LIN {X 75.422,Y -35.957,Z -72.523,A -90.000,B 90.000,C 0.000} C_DIS
LIN {X 75.798,Y -35.942,Z -72.914,A -90.000,B 90.000,C 0.000} C_DIS
LIN {X 76.219,Y -35.930,Z -73.360,A -90.000,B 90.000,C 0.000} C_DIS
LIN {X 76.678,Y -35.924,Z -73.869,A -90.000,B 90.000,C 0.000} C_DIS
LIN {X 76.731,Y -35.865,Z -73.840,A -90.000,B 90.000,C 0.000} C_DIS
LIN {X 76.810,Y -35.794,Z -73.827,A -90.000,B 90.000,C 0.000} C_DIS
LIN {X 76.846,Y -35.765,Z -73.824,A -90.000,B 90.000,C 0.000} C_DIS
LIN {X 77.170,Y -35.545,Z -73.872,A -90.000,B 90.000,C 0.000} C_DIS
LIN {X 77.258,Y -35.499,Z -73.909,A -90.000,B 90.000,C 0.000} C_DIS
LIN {X 77.415,Y -35.431,Z -73.994,A -90.000,B 90.000,C 0.000} C_DIS
LIN {X 77.609,Y -35.368,Z -74.129,A -90.000,B 90.000,C 0.000} C_DIS
LIN {X 77.655,Y -35.356,Z -74.166,A -90.000,B 90.000,C 0.000} C_DIS
LIN {X 77.754,Y -35.347,Z -73.596,A -90.000,B 90.000,C 0.000} C_DIS
LIN {X 77.829,Y -35.339,Z -73.246,A -90.000,B 90.000,C 0.000} C_DIS
LIN {X 78.002,Y -35.325,Z -72.470,A -90.000,B 90.000,C 0.000} C_DIS
LIN {X 78.095,Y -35.319,Z -72.097,A -90.000,B 90.000,C 0.000} C_DIS
LIN {X 78.171,Y -35.317,Z -71.800,A -90.000,B 90.000,C 0.000} C_DIS
LIN {X 78.247,Y -35.314,Z -71.562,A -90.000,B 90.000,C 0.000} C_DIS
LIN {X 78.534,Y -35.309,Z -70.687,A -90.000,B 90.000,C 0.000} C_DIS
LIN {X 78.778,Y -35.308,Z -69.955,A -90.000,B 90.000,C 0.000} C_DIS
LIN {X 78.789,Y -36.719,Z -69.922,A -90.000,B 90.000,C 0.000} C_DIS
LIN {X 78.791,Y -36.729,Z -69.917,A -90.000,B 90.000,C 0.000} C_DIS
LIN {X 78.792,Y -36.756,Z -69.913,A -90.000,B 90.000,C 0.000} C_DIS
LIN {X 78.804,Y -35.308,Z -69.881,A -90.000,B 90.000,C 0.000} C_DIS
LIN {X 79.057,Y -35.310,Z -69.150,A -90.000,B 90.000,C 0.000} C_DIS
LIN {X 79.142,Y -35.308,Z -68.907,A -90.000,B 90.000,C 0.000} C_DIS
LIN {X 79.365,Y -35.304,Z -68.248,A -90.000,B 90.000,C 0.000} C_DIS
LIN {X 79.416,Y -35.303,Z -68.080,A -90.000,B 90.000,C 0.000} C_DIS
LIN {X 79.428,Y -35.303,Z -68.032,A -90.000,B 90.000,C 0.000} C_DIS
LIN {X 79.454,Y -35.306,Z -67.989,A -90.000,B 90.000,C 0.000} C_DIS
LIN {X 79.532,Y -35.307,Z -67.831,A -90.000,B 90.000,C 0.000} C_DIS
LIN {X 79.818,Y -35.308,Z -67.197,A -90.000,B 90.000,C 0.000} C_DIS
LIN {X 79.922,Y -35.308,Z -66.959,A -90.000,B 90.000,C 0.000} C_DIS
LIN {X 79.922,Y -60.000,Z -66.959,A -90.000,B 90.000,C 0.000} C_DIS
LIN {X 89.581,Y -60.000,Z -54.050,A -90.000,B 90.000,C 0.000} C_DIS
LIN {X 89.581,Y -35.308,Z -54.050,A -90.000,B 90.000,C 0.000} C_DIS
LIN {X 89.698,Y -35.308,Z -53.943,A -90.000,B 90.000,C 0.000} C_DIS
LIN {X 89.987,Y -35.308,Z -53.665,A -90.000,B 90.000,C 0.000} C_DIS
LIN {X 90.272,Y -35.308,Z -53.420,A -90.000,B 90.000,C 0.000} C_DIS
LIN {X 91.215,Y -35.306,Z -52.572,A -90.000,B 90.000,C 0.000} C_DIS
LIN {X 91.916,Y -35.303,Z -51.957,A -90.000,B 90.000,C 0.000} C_DIS
LIN {X 92.305,Y -35.300,Z -51.627,A -90.000,B 90.000,C 0.000} C_DIS
LIN {X 92.595,Y -35.296,Z -51.392,A -90.000,B 90.000,C 0.000} C_DIS
LIN {X 92.801,Y -35.293,Z -51.238,A -90.000,B 90.000,C 0.000} C_DIS
LIN {X 92.938,Y -35.289,Z -51.149,A -90.000,B 90.000,C 0.000} C_DIS
LIN {X 92.966,Y -35.286,Z -51.121,A -90.000,B 90.000,C 0.000} C_DIS
LIN {X 92.990,Y -35.285,Z -51.107,A -90.000,B 90.000,C 0.000} C_DIS
LIN {X 92.992,Y -46.259,Z -51.106,A -90.000,B 90.000,C 0.000} C_DIS
LIN {X 92.993,Y -46.306,Z -51.106,A -90.000,B 90.000,C 0.000} C_DIS
LIN {X 93.018,Y -46.533,Z -51.097,A -90.000,B 90.000,C 0.000} C_DIS
LIN {X 93.039,Y -46.657,Z -51.092,A -90.000,B 90.000,C 0.000} C_DIS
LIN {X 93.071,Y -46.842,Z -51.092,A -90.000,B 90.000,C 0.000} C_DIS
LIN {X 93.093,Y -46.989,Z -51.102,A -90.000,B 90.000,C 0.000} C_DIS
LIN {X 93.119,Y -47.185,Z -51.127,A -90.000,B 90.000,C 0.000} C_DIS
LIN {X 93.133,Y -47.246,Z -51.132,A -90.000,B 90.000,C 0.000} C_DIS
LIN {X 93.143,Y -47.273,Z -51.131,A -90.000,B 90.000,C 0.000} C_DIS
LIN {X 93.155,Y -47.296,Z -51.128,A -90.000,B 90.000,C 0.000} C_DIS
LIN {X 93.171,Y -47.316,Z -51.121,A -90.000,B 90.000,C 0.000} C_DIS
LIN {X 93.191,Y -47.332,Z -51.111,A -90.000,B 90.000,C 0.000} C_DIS
LIN {X 93.215,Y -47.345,Z -51.095,A -90.000,B 90.000,C 0.000} C_DIS
LIN {X 93.244,Y -47.355,Z -51.075,A -90.000,B 90.000,C 0.000} C_DIS
LIN {X 93.279,Y -47.360,Z -51.049,A -90.000,B 90.000,C 0.000} C_DIS
LIN {X 93.321,Y -47.361,Z -51.017,A -90.000,B 90.000,C 0.000} C_DIS
LIN {X 93.424,Y -47.351,Z -50.931,A -90.000,B 90.000,C 0.000} C_DIS
LIN {X 93.559,Y -47.320,Z -50.814,A -90.000,B 90.000,C 0.000} C_DIS
LIN {X 93.733,Y -47.264,Z -50.658,A -90.000,B 90.000,C 0.000} C_DIS
LIN {X 93.948,Y -47.178,Z -50.461,A -90.000,B 90.000,C 0.000} C_DIS
LIN {X 94.208,Y -47.057,Z -50.218,A -90.000,B 90.000,C 0.000} C_DIS
LIN {X 94.519,Y -46.887,Z -49.925,A -90.000,B 90.000,C 0.000} C_DIS
LIN {X 94.884,Y -46.660,Z -49.576,A -90.000,B 90.000,C 0.000} C_DIS
LIN {X 95.309,Y -46.351,Z -49.169,A -90.000,B 90.000,C 0.000} C_DIS
LIN {X 95.545,Y -46.143,Z -48.941,A -90.000,B 90.000,C 0.000} C_DIS
LIN {X 95.670,Y -46.013,Z -48.821,A -90.000,B 90.000,C 0.000} C_DIS
LIN {X 95.798,Y -45.845,Z -48.697,A -90.000,B 90.000,C 0.000} C_DIS
LIN {X 95.864,Y -45.722,Z -48.633,A -90.000,B 90.000,C 0.000} C_DIS
LIN {X 95.897,Y -45.614,Z -48.601,A -90.000,B 90.000,C 0.000} C_DIS
LIN {X 95.904,Y -45.562,Z -48.595,A -90.000,B 90.000,C 0.000} C_DIS
LIN {X 95.906,Y -35.302,Z -48.593,A -90.000,B 90.000,C 0.000} C_DIS
LIN {X 96.069,Y -35.303,Z -48.437,A -90.000,B 90.000,C 0.000} C_DIS
LIN {X 96.365,Y -35.308,Z -48.166,A -90.000,B 90.000,C 0.000} C_DIS
LIN {X 96.504,Y -35.310,Z -48.031,A -90.000,B 90.000,C 0.000} C_DIS
LIN {X 96.976,Y -35.308,Z -47.573,A -90.000,B 90.000,C 0.000} C_DIS
LIN {X 96.976,Y -60.000,Z -47.573,A -90.000,B 90.000,C 0.000} C_DIS
LIN {X -13.596,Y -60.000,Z -67.623,A -90.000,B 90.000,C 0.000} C_DIS
LIN {X -13.596,Y -35.308,Z -67.623,A -90.000,B 90.000,C 0.000} C_DIS
LIN {X -12.574,Y -35.360,Z -67.585,A -90.000,B 90.000,C 0.000} C_DIS
LIN {X -12.388,Y -35.371,Z -67.585,A -90.000,B 90.000,C 0.000} C_DIS
LIN {X -11.858,Y -35.405,Z -67.599,A -90.000,B 90.000,C 0.000} C_DIS
LIN {X -11.441,Y -35.437,Z -67.609,A -90.000,B 90.000,C 0.000} C_DIS
LIN {X -10.549,Y -35.505,Z -67.647,A -90.000,B 90.000,C 0.000} C_DIS
LIN {X -8.614,Y -35.635,Z -67.743,A -90.000,B 90.000,C 0.000} C_DIS
LIN {X -8.402,Y -35.650,Z -67.760,A -90.000,B 90.000,C 0.000} C_DIS
LIN {X -7.555,Y -35.711,Z -67.851,A -90.000,B 90.000,C 0.000} C_DIS
LIN {X -6.626,Y -35.780,Z -67.956,A -90.000,B 90.000,C 0.000} C_DIS
LIN {X -5.314,Y -35.895,Z -68.093,A -90.000,B 90.000,C 0.000} C_DIS
LIN {X -4.465,Y -35.968,Z -68.175,A -90.000,B 90.000,C 0.000} C_DIS
LIN {X -4.298,Y -35.983,Z -68.196,A -90.000,B 90.000,C 0.000} C_DIS
LIN {X -3.714,Y -36.037,Z -68.287,A -90.000,B 90.000,C 0.000} C_DIS
LIN {X -2.584,Y -36.140,Z -68.444,A -90.000,B 90.000,C 0.000} C_DIS
LIN {X -2.065,Y -36.205,Z -68.510,A -90.000,B 90.000,C 0.000} C_DIS
LIN {X -1.663,Y -36.251,Z -68.557,A -90.000,B 90.000,C 0.000} C_DIS
LIN {X -0.777,Y -36.350,Z -68.643,A -90.000,B 90.000,C 0.000} C_DIS
LIN {X 0.304,Y -36.461,Z -68.748,A -90.000,B 90.000,C 0.000} C_DIS
LIN {X 0.445,Y -36.476,Z -68.766,A -90.000,B 90.000,C 0.000} C_DIS
LIN {X 1.033,Y -36.542,Z -68.853,A -90.000,B 90.000,C 0.000} C_DIS
LIN {X 1.072,Y -36.545,Z -68.853,A -90.000,B 90.000,C 0.000} C_DIS
LIN {X 1.180,Y -36.530,Z -68.728,A -90.000,B 90.000,C 0.000} C_DIS
LIN {X 1.354,Y -36.514,Z -68.541,A -90.000,B 90.000,C 0.000} C_DIS
LIN {X 1.487,Y -36.499,Z -68.410,A -90.000,B 90.000,C 0.000} C_DIS
LIN {X 1.693,Y -36.460,Z -68.221,A -90.000,B 90.000,C 0.000} C_DIS
LIN {X 1.761,Y -36.448,Z -68.160,A -90.000,B 90.000,C 0.000} C_DIS
LIN {X 1.873,Y -36.431,Z -68.070,A -90.000,B 90.000,C 0.000} C_DIS
LIN {X 2.044,Y -36.406,Z -67.940,A -90.000,B 90.000,C 0.000} C_DIS
LIN {X 2.234,Y -36.380,Z -67.806,A -90.000,B 90.000,C 0.000} C_DIS
LIN {X 2.406,Y -36.357,Z -67.692,A -90.000,B 90.000,C 0.000} C_DIS
LIN {X 2.639,Y -36.329,Z -67.546,A -90.000,B 90.000,C 0.000} C_DIS
LIN {X 2.812,Y -36.305,Z -67.428,A -90.000,B 90.000,C 0.000} C_DIS
LIN {X 3.276,Y -36.201,Z -67.126,A -90.000,B 90.000,C 0.000} C_DIS
LIN {X 3.444,Y -36.166,Z -67.024,A -90.000,B 90.000,C 0.000} C_DIS
LIN {X 3.614,Y -36.134,Z -66.931,A -90.000,B 90.000,C 0.000} C_DIS
LIN {X 3.853,Y -36.097,Z -66.819,A -90.000,B 90.000,C 0.000} C_DIS
LIN {X 3.948,Y -36.084,Z -66.778,A -90.000,B 90.000,C 0.000} C_DIS
LIN {X 4.233,Y -36.047,Z -66.662,A -90.000,B 90.000,C 0.000} C_DIS
LIN {X 4.353,Y -36.033,Z -66.617,A -90.000,B 90.000,C 0.000} C_DIS
LIN {X 4.683,Y -36.009,Z -66.505,A -90.000,B 90.000,C 0.000} C_DIS
LIN {X 4.875,Y -35.985,Z -66.444,A -90.000,B 90.000,C 0.000} C_DIS
LIN {X 5.852,Y -35.847,Z -66.145,A -90.000,B 90.000,C 0.000} C_DIS
LIN {X 6.202,Y -35.800,Z -66.046,A -90.000,B 90.000,C 0.000} C_DIS
LIN {X 6.435,Y -35.772,Z -65.986,A -90.000,B 90.000,C 0.000} C_DIS
LIN {X 6.689,Y -35.747,Z -65.930,A -90.000,B 90.000,C 0.000} C_DIS
LIN {X 6.738,Y -35.742,Z -65.921,A -90.000,B 90.000,C 0.000} C_DIS
LIN {X 7.225,Y -35.706,Z -65.832,A -90.000,B 90.000,C 0.000} C_DIS
LIN {X 7.523,Y -35.685,Z -65.777,A -90.000,B 90.000,C 0.000} C_DIS
LIN {X 7.613,Y -35.680,Z -65.763,A -90.000,B 90.000,C 0.000} C_DIS
LIN {X 7.872,Y -35.669,Z -65.728,A -90.000,B 90.000,C 0.000} C_DIS
LIN {X 8.114,Y -35.663,Z -65.702,A -90.000,B 90.000,C 0.000} C_DIS
LIN {X 8.854,Y -35.619,Z -65.637,A -90.000,B 90.000,C 0.000} C_DIS
LIN {X 9.243,Y -35.584,Z -65.608,A -90.000,B 90.000,C 0.000} C_DIS
LIN {X 9.497,Y -35.559,Z -65.590,A -90.000,B 90.000,C 0.000} C_DIS
LIN {X 9.712,Y -35.542,Z -65.579,A -90.000,B 90.000,C 0.000} C_DIS
LIN {X 9.853,Y -35.535,Z -65.579,A -90.000,B 90.000,C 0.000} C_DIS
LIN {X 10.047,Y -35.527,Z -65.583,A -90.000,B 90.000,C 0.000} C_DIS
LIN {X 10.154,Y -35.524,Z -65.588,A -90.000,B 90.000,C 0.000} C_DIS
LIN {X 10.498,Y -35.522,Z -65.612,A -90.000,B 90.000,C 0.000} C_DIS
LIN {X 10.799,Y -35.527,Z -65.640,A -90.000,B 90.000,C 0.000} C_DIS
LIN {X 10.993,Y -35.530,Z -65.659,A -90.000,B 90.000,C 0.000} C_DIS
LIN {X 11.036,Y -35.530,Z -65.664,A -90.000,B 90.000,C 0.000} C_DIS
LIN {X 11.092,Y -35.487,Z -65.606,A -90.000,B 90.000,C 0.000} C_DIS
LIN {X 11.178,Y -35.423,Z -65.522,A -90.000,B 90.000,C 0.000} C_DIS
LIN {X 11.344,Y -35.308,Z -65.374,A -90.000,B 90.000,C 0.000} C_DIS
LIN {X 11.344,Y -60.000,Z -65.374,A -90.000,B 90.000,C 0.000} C_DIS
LIN {X -10.557,Y -60.000,Z -65.654,A -90.000,B 90.000,C 0.000} C_DIS
LIN {X -10.557,Y -35.308,Z -65.654,A -90.000,B 90.000,C 0.000} C_DIS
LIN {X -10.015,Y -35.339,Z -65.681,A -90.000,B 90.000,C 0.000} C_DIS
LIN {X -8.500,Y -35.403,Z -65.760,A -90.000,B 90.000,C 0.000} C_DIS
LIN {X -8.411,Y -35.409,Z -65.774,A -90.000,B 90.000,C 0.000} C_DIS
LIN {X -8.173,Y -35.418,Z -65.786,A -90.000,B 90.000,C 0.000} C_DIS
LIN {X -7.110,Y -35.475,Z -65.905,A -90.000,B 90.000,C 0.000} C_DIS
LIN {X -6.382,Y -35.515,Z -65.989,A -90.000,B 90.000,C 0.000} C_DIS
LIN {X -6.093,Y -35.531,Z -66.021,A -90.000,B 90.000,C 0.000} C_DIS
LIN {X -5.091,Y -35.594,Z -66.128,A -90.000,B 90.000,C 0.000} C_DIS
LIN {X -4.180,Y -35.637,Z -66.223,A -90.000,B 90.000,C 0.000} C_DIS
LIN {X -3.966,Y -35.649,Z -66.253,A -90.000,B 90.000,C 0.000} C_DIS
LIN {X -3.387,Y -35.686,Z -66.345,A -90.000,B 90.000,C 0.000} C_DIS
LIN {X -2.118,Y -35.760,Z -66.529,A -90.000,B 90.000,C 0.000} C_DIS
LIN {X -1.766,Y -35.791,Z -66.576,A -90.000,B 90.000,C 0.000} C_DIS
LIN {X -1.433,Y -35.819,Z -66.618,A -90.000,B 90.000,C 0.000} C_DIS
LIN {X 0.371,Y -35.957,Z -66.806,A -90.000,B 90.000,C 0.000} C_DIS
LIN {X 0.430,Y -35.942,Z -66.757,A -90.000,B 90.000,C 0.000} C_DIS
LIN {X 0.581,Y -35.905,Z -66.636,A -90.000,B 90.000,C 0.000} C_DIS
LIN {X 0.657,Y -35.887,Z -66.577,A -90.000,B 90.000,C 0.000} C_DIS
LIN {X 0.888,Y -35.824,Z -66.415,A -90.000,B 90.000,C 0.000} C_DIS
LIN {X 1.126,Y -35.764,Z -66.259,A -90.000,B 90.000,C 0.000} C_DIS
LIN {X 1.345,Y -35.703,Z -66.128,A -90.000,B 90.000,C 0.000} C_DIS
LIN {X 1.553,Y -35.649,Z -66.010,A -90.000,B 90.000,C 0.000} C_DIS
LIN {X 2.067,Y -35.517,Z -65.684,A -90.000,B 90.000,C 0.000} C_DIS
LIN {X 2.150,Y -35.495,Z -65.632,A -90.000,B 90.000,C 0.000} C_DIS
LIN {X 2.435,Y -35.413,Z -65.470,A -90.000,B 90.000,C 0.000} C_DIS
LIN {X 2.662,Y -35.355,Z -65.354,A -90.000,B 90.000,C 0.000} C_DIS
LIN {X 2.841,Y -35.308,Z -65.277,A -90.000,B 90.000,C 0.000} C_DIS
LIN {X 2.841,Y -60.000,Z -65.277,A -90.000,B 90.000,C 0.000} C_DIS
LIN {X -38.882,Y -60.000,Z -100.616,A -90.000,B 90.000,C 0.000} C_DIS
LIN {X -38.882,Y -35.308,Z -100.616,A -90.000,B 90.000,C 0.000} C_DIS
LIN {X -38.869,Y -35.369,Z -100.386,A -90.000,B 90.000,C 0.000} C_DIS
LIN {X -38.831,Y -35.507,Z -99.867,A -90.000,B 90.000,C 0.000} C_DIS
LIN {X -38.799,Y -35.593,Z -99.544,A -90.000,B 90.000,C 0.000} C_DIS
LIN {X -38.749,Y -35.706,Z -99.117,A -90.000,B 90.000,C 0.000} C_DIS
LIN {X -38.638,Y -35.920,Z -98.326,A -90.000,B 90.000,C 0.000} C_DIS
LIN {X -38.842,Y -35.915,Z -98.047,A -90.000,B 90.000,C 0.000} C_DIS
LIN {X -39.961,Y -35.875,Z -96.572,A -90.000,B 90.000,C 0.000} C_DIS
LIN {X -40.111,Y -35.870,Z -96.357,A -90.000,B 90.000,C 0.000} C_DIS
LIN {X -40.365,Y -35.864,Z -95.966,A -90.000,B 90.000,C 0.000} C_DIS
LIN {X -40.440,Y -35.864,Z -95.843,A -90.000,B 90.000,C 0.000} C_DIS
LIN {X -41.255,Y -35.872,Z -94.460,A -90.000,B 90.000,C 0.000} C_DIS
LIN {X -41.491,Y -35.873,Z -94.057,A -90.000,B 90.000,C 0.000} C_DIS
LIN {X -41.725,Y -35.878,Z -93.628,A -90.000,B 90.000,C 0.000} C_DIS
LIN {X -41.850,Y -35.882,Z -93.380,A -90.000,B 90.000,C 0.000} C_DIS
LIN {X -42.234,Y -35.885,Z -92.604,A -90.000,B 90.000,C 0.000} C_DIS
LIN {X -42.654,Y -35.888,Z -91.745,A -90.000,B 90.000,C 0.000} C_DIS
LIN {X -42.697,Y -35.890,Z -91.651,A -90.000,B 90.000,C 0.000} C_DIS
LIN {X -42.806,Y -35.896,Z -91.395,A -90.000,B 90.000,C 0.000} C_DIS
LIN {X -43.104,Y -35.925,Z -90.590,A -90.000,B 90.000,C 0.000} C_DIS
LIN {X -43.341,Y -35.949,Z -89.883,A -90.000,B 90.000,C 0.000} C_DIS
LIN {X -43.362,Y -35.951,Z -89.813,A -90.000,B 90.000,C 0.000} C_DIS
LIN {X -43.528,Y -35.973,Z -89.234,A -90.000,B 90.000,C 0.000} C_DIS
LIN {X -43.715,Y -35.988,Z -88.558,A -90.000,B 90.000,C 0.000} C_DIS
LIN {X -43.878,Y -36.004,Z -87.941,A -90.000,B 90.000,C 0.000} C_DIS
LIN {X -43.939,Y -36.013,Z -87.662,A -90.000,B 90.000,C 0.000} C_DIS
LIN {X -44.014,Y -36.027,Z -87.293,A -90.000,B 90.000,C 0.000} C_DIS
LIN {X -44.048,Y -36.036,Z -87.101,A -90.000,B 90.000,C 0.000} C_DIS
LIN {X -44.083,Y -36.050,Z -86.869,A -90.000,B 90.000,C 0.000} C_DIS
LIN {X -44.095,Y -36.057,Z -86.764,A -90.000,B 90.000,C 0.000} C_DIS
LIN {X -44.121,Y -36.079,Z -86.489,A -90.000,B 90.000,C 0.000} C_DIS
LIN {X -44.141,Y -36.110,Z -85.867,A -90.000,B 90.000,C 0.000} C_DIS
LIN {X -44.183,Y -36.168,Z -84.334,A -90.000,B 90.000,C 0.000} C_DIS
LIN {X -44.182,Y -36.178,Z -84.112,A -90.000,B 90.000,C 0.000} C_DIS
LIN {X -44.177,Y -36.178,Z -84.012,A -90.000,B 90.000,C 0.000} C_DIS
LIN {X -44.146,Y -36.182,Z -83.590,A -90.000,B 90.000,C 0.000} C_DIS
LIN {X -44.132,Y -36.185,Z -83.490,A -90.000,B 90.000,C 0.000} C_DIS
LIN {X -44.070,Y -36.198,Z -83.103,A -90.000,B 90.000,C 0.000} C_DIS
LIN {X -43.808,Y -36.261,Z -81.992,A -90.000,B 90.000,C 0.000} C_DIS
LIN {X -43.696,Y -36.270,Z -81.536,A -90.000,B 90.000,C 0.000} C_DIS
LIN {X -43.643,Y -36.273,Z -81.324,A -90.000,B 90.000,C 0.000} C_DIS
LIN {X -43.570,Y -36.276,Z -81.023,A -90.000,B 90.000,C 0.000} C_DIS
LIN {X -43.479,Y -36.284,Z -80.710,A -90.000,B 90.000,C 0.000} C_DIS
LIN {X -43.422,Y -36.288,Z -80.544,A -90.000,B 90.000,C 0.000} C_DIS
LIN {X -43.347,Y -36.296,Z -80.340,A -90.000,B 90.000,C 0.000} C_DIS
LIN {X -43.287,Y -36.303,Z -80.195,A -90.000,B 90.000,C 0.000} C_DIS
LIN {X -43.190,Y -36.315,Z -79.973,A -90.000,B 90.000,C 0.000} C_DIS
LIN {X -42.919,Y -36.335,Z -79.364,A -90.000,B 90.000,C 0.000} C_DIS
LIN {X -42.740,Y -36.346,Z -78.963,A -90.000,B 90.000,C 0.000} C_DIS
LIN {X -42.457,Y -36.355,Z -78.338,A -90.000,B 90.000,C 0.000} C_DIS
LIN {X -42.313,Y -36.363,Z -78.065,A -90.000,B 90.000,C 0.000} C_DIS
LIN {X -42.234,Y -36.367,Z -77.922,A -90.000,B 90.000,C 0.000} C_DIS
LIN {X -42.046,Y -36.379,Z -77.603,A -90.000,B 90.000,C 0.000} C_DIS
LIN {X -41.973,Y -36.384,Z -77.488,A -90.000,B 90.000,C 0.000} C_DIS
LIN {X -41.159,Y -36.424,Z -76.230,A -90.000,B 90.000,C 0.000} C_DIS
LIN {X -40.955,Y -36.432,Z -75.918,A -90.000,B 90.000,C 0.000} C_DIS
LIN {X -40.124,Y -36.468,Z -74.740,A -90.000,B 90.000,C 0.000} C_DIS
LIN {X -40.001,Y -36.473,Z -74.579,A -90.000,B 90.000,C 0.000} C_DIS
LIN {X -39.792,Y -36.478,Z -74.328,A -90.000,B 90.000,C 0.000} C_DIS
LIN {X -39.294,Y -36.483,Z -73.741,A -90.000,B 90.000,C 0.000} C_DIS
LIN {X -39.128,Y -36.485,Z -73.549,A -90.000,B 90.000,C 0.000} C_DIS
LIN {X -38.976,Y -36.489,Z -73.388,A -90.000,B 90.000,C 0.000} C_DIS
LIN {X -38.463,Y -36.497,Z -72.873,A -90.000,B 90.000,C 0.000} C_DIS
LIN {X -38.273,Y -36.492,Z -72.698,A -90.000,B 90.000,C 0.000} C_DIS
LIN {X -37.803,Y -36.487,Z -72.303,A -90.000,B 90.000,C 0.000} C_DIS
LIN {X -37.366,Y -36.479,Z -71.939,A -90.000,B 90.000,C 0.000} C_DIS
LIN {X -36.855,Y -36.466,Z -71.517,A -90.000,B 90.000,C 0.000} C_DIS
LIN {X -36.651,Y -36.463,Z -71.360,A -90.000,B 90.000,C 0.000} C_DIS
LIN {X -36.555,Y -36.462,Z -71.288,A -90.000,B 90.000,C 0.000} C_DIS
LIN {X -36.426,Y -36.462,Z -71.201,A -90.000,B 90.000,C 0.000} C_DIS
LIN {X -36.251,Y -36.454,Z -71.089,A -90.000,B 90.000,C 0.000} C_DIS
LIN {X -36.112,Y -36.449,Z -71.009,A -90.000,B 90.000,C 0.000} C_DIS
LIN {X -35.987,Y -36.445,Z -70.944,A -90.000,B 90.000,C 0.000} C_DIS
LIN {X -35.881,Y -36.441,Z -70.890,A -90.000,B 90.000,C 0.000} C_DIS
LIN {X -35.610,Y -36.435,Z -70.766,A -90.000,B 90.000,C 0.000} C_DIS
LIN {X -35.409,Y -36.426,Z -70.678,A -90.000,B 90.000,C 0.000} C_DIS
LIN {X -35.266,Y -36.421,Z -70.620,A -90.000,B 90.000,C 0.000} C_DIS
LIN {X -34.462,Y -36.396,Z -70.308,A -90.000,B 90.000,C 0.000} C_DIS
LIN {X -33.940,Y -36.373,Z -70.109,A -90.000,B 90.000,C 0.000} C_DIS
LIN {X -33.750,Y -36.367,Z -70.045,A -90.000,B 90.000,C 0.000} C_DIS
LIN {X -33.023,Y -36.353,Z -69.835,A -90.000,B 90.000,C 0.000} C_DIS
LIN {X -32.640,Y -36.341,Z -69.726,A -90.000,B 90.000,C 0.000} C_DIS
LIN {X -32.463,Y -36.332,Z -69.681,A -90.000,B 90.000,C 0.000} C_DIS
LIN {X -32.083,Y -36.313,Z -69.601,A -90.000,B 90.000,C 0.000} C_DIS
LIN {X -31.626,Y -36.272,Z -69.514,A -90.000,B 90.000,C 0.000} C_DIS
LIN {X -31.454,Y -36.259,Z -69.488,A -90.000,B 90.000,C 0.000} C_DIS
LIN {X -31.282,Y -36.247,Z -69.465,A -90.000,B 90.000,C 0.000} C_DIS
LIN {X -31.014,Y -36.233,Z -69.441,A -90.000,B 90.000,C 0.000} C_DIS
LIN {X -30.534,Y -36.207,Z -69.402,A -90.000,B 90.000,C 0.000} C_DIS
LIN {X -29.760,Y -36.158,Z -69.343,A -90.000,B 90.000,C 0.000} C_DIS
LIN {X -29.603,Y -36.147,Z -69.338,A -90.000,B 90.000,C 0.000} C_DIS
LIN {X -29.336,Y -36.132,Z -69.339,A -90.000,B 90.000,C 0.000} C_DIS
LIN {X -28.844,Y -36.108,Z -69.351,A -90.000,B 90.000,C 0.000} C_DIS
LIN {X -28.657,Y -36.100,Z -69.363,A -90.000,B 90.000,C 0.000} C_DIS
LIN {X -28.473,Y -36.094,Z -69.379,A -90.000,B 90.000,C 0.000} C_DIS
LIN {X -28.192,Y -36.090,Z -69.420,A -90.000,B 90.000,C 0.000} C_DIS
LIN {X -28.046,Y -36.089,Z -69.446,A -90.000,B 90.000,C 0.000} C_DIS
LIN {X -28.006,Y -36.090,Z -69.454,A -90.000,B 90.000,C 0.000} C_DIS
LIN {X -27.651,Y -36.087,Z -69.512,A -90.000,B 90.000,C 0.000} C_DIS
LIN {X -26.416,Y -36.047,Z -69.723,A -90.000,B 90.000,C 0.000} C_DIS
LIN {X -26.245,Y -36.039,Z -69.754,A -90.000,B 90.000,C 0.000} C_DIS
LIN {X -25.938,Y -36.029,Z -69.818,A -90.000,B 90.000,C 0.000} C_DIS
LIN {X -25.687,Y -36.024,Z -69.880,A -90.000,B 90.000,C 0.000} C_DIS
LIN {X -25.522,Y -36.023,Z -69.926,A -90.000,B 90.000,C 0.000} C_DIS
LIN {X -24.759,Y -35.999,Z -70.092,A -90.000,B 90.000,C 0.000} C_DIS
LIN {X -24.434,Y -35.984,Z -70.165,A -90.000,B 90.000,C 0.000} C_DIS
LIN {X -23.889,Y -35.947,Z -70.259,A -90.000,B 90.000,C 0.000} C_DIS
LIN {X -23.667,Y -35.868,Z -70.143,A -90.000,B 90.000,C 0.000} C_DIS
LIN {X -23.431,Y -35.788,Z -70.016,A -90.000,B 90.000,C 0.000} C_DIS
LIN {X -23.249,Y -35.725,Z -69.922,A -90.000,B 90.000,C 0.000} C_DIS
LIN {X -23.142,Y -35.689,Z -69.871,A -90.000,B 90.000,C 0.000} C_DIS
LIN {X -23.071,Y -35.662,Z -69.840,A -90.000,B 90.000,C 0.000} C_DIS
LIN {X -22.773,Y -35.559,Z -69.727,A -90.000,B 90.000,C 0.000} C_DIS
LIN {X -22.534,Y -35.477,Z -69.640,A -90.000,B 90.000,C 0.000} C_DIS
LIN {X -22.196,Y -35.354,Z -69.521,A -90.000,B 90.000,C 0.000} C_DIS
LIN {X -22.139,Y -35.333,Z -69.502,A -90.000,B 90.000,C 0.000} C_DIS
LIN {X -22.058,Y -35.308,Z -69.472,A -90.000,B 90.000,C 0.000} C_DIS
LIN {X -22.058,Y -60.000,Z -69.472,A -90.000,B 90.000,C 0.000} C_DIS
LIN {X -45.910,Y -60.000,Z -87.224,A -90.000,B 90.000,C 0.000} C_DIS
LIN {X -45.910,Y -35.308,Z -87.224,A -90.000,B 90.000,C 0.000} C_DIS
LIN {X -45.947,Y -35.321,Z -86.940,A -90.000,B 90.000,C 0.000} C_DIS
LIN {X -45.973,Y -35.338,Z -86.640,A -90.000,B 90.000,C 0.000} C_DIS
LIN {X -45.982,Y -35.347,Z -86.499,A -90.000,B 90.000,C 0.000} C_DIS
LIN {X -46.018,Y -35.411,Z -85.654,A -90.000,B 90.000,C 0.000} C_DIS
LIN {X -46.045,Y -35.461,Z -85.027,A -90.000,B 90.000,C 0.000} C_DIS
LIN {X -46.063,Y -35.488,Z -84.298,A -90.000,B 90.000,C 0.000} C_DIS
LIN {X -46.062,Y -35.500,Z -84.020,A -90.000,B 90.000,C 0.000} C_DIS
LIN {X -46.056,Y -35.510,Z -83.852,A -90.000,B 90.000,C 0.000} C_DIS
LIN {X -46.032,Y -35.536,Z -83.442,A -90.000,B 90.000,C 0.000} C_DIS
LIN {X -46.011,Y -35.553,Z -83.223,A -90.000,B 90.000,C 0.000} C_DIS
LIN {X -45.955,Y -35.589,Z -82.828,A -90.000,B 90.000,C 0.000} C_DIS
LIN {X -45.935,Y -35.594,Z -82.707,A -90.000,B 90.000,C 0.000} C_DIS
LIN {X -45.873,Y -35.610,Z -82.438,A -90.000,B 90.000,C 0.000} C_DIS
LIN {X -45.494,Y -35.704,Z -80.820,A -90.000,B 90.000,C 0.000} C_DIS
LIN {X -45.433,Y -35.708,Z -80.567,A -90.000,B 90.000,C 0.000} C_DIS
LIN {X -45.408,Y -35.710,Z -80.475,A -90.000,B 90.000,C 0.000} C_DIS
LIN {X -45.292,Y -35.721,Z -80.081,A -90.000,B 90.000,C 0.000} C_DIS
LIN {X -45.218,Y -35.730,Z -79.863,A -90.000,B 90.000,C 0.000} C_DIS
LIN {X -45.114,Y -35.743,Z -79.582,A -90.000,B 90.000,C 0.000} C_DIS
LIN {X -45.006,Y -35.759,Z -79.326,A -90.000,B 90.000,C 0.000} C_DIS
LIN {X -44.833,Y -35.786,Z -78.927,A -90.000,B 90.000,C 0.000} C_DIS
LIN {X -44.634,Y -35.806,Z -78.477,A -90.000,B 90.000,C 0.000} C_DIS
LIN {X -44.214,Y -35.834,Z -77.536,A -90.000,B 90.000,C 0.000} C_DIS
LIN {X -44.159,Y -35.839,Z -77.424,A -90.000,B 90.000,C 0.000} C_DIS
LIN {X -43.999,Y -35.854,Z -77.117,A -90.000,B 90.000,C 0.000} C_DIS
LIN {X -43.894,Y -35.863,Z -76.927,A -90.000,B 90.000,C 0.000} C_DIS
LIN {X -43.670,Y -35.877,Z -76.549,A -90.000,B 90.000,C 0.000} C_DIS
LIN {X -43.046,Y -35.924,Z -75.575,A -90.000,B 90.000,C 0.000} C_DIS
LIN {X -42.574,Y -35.949,Z -74.848,A -90.000,B 90.000,C 0.000} C_DIS
LIN {X -42.191,Y -35.974,Z -74.300,A -90.000,B 90.000,C 0.000} C_DIS
LIN {X -41.847,Y -35.989,Z -73.810,A -90.000,B 90.000,C 0.000} C_DIS
LIN {X -41.660,Y -35.992,Z -73.550,A -90.000,B 90.000,C 0.000} C_DIS
LIN {X -41.490,Y -35.997,Z -73.332,A -90.000,B 90.000,C 0.000} C_DIS
LIN {X -41.148,Y -36.010,Z -72.921,A -90.000,B 90.000,C 0.000} C_DIS
LIN {X -40.759,Y -36.019,Z -72.460,A -90.000,B 90.000,C 0.000} C_DIS
LIN {X -40.585,Y -36.024,Z -72.259,A -90.000,B 90.000,C 0.000} C_DIS
LIN {X -40.402,Y -36.026,Z -72.065,A -90.000,B 90.000,C 0.000} C_DIS
LIN {X -39.837,Y -36.021,Z -71.499,A -90.000,B 90.000,C 0.000} C_DIS
LIN {X -39.596,Y -36.018,Z -71.275,A -90.000,B 90.000,C 0.000} C_DIS
LIN {X -39.526,Y -36.018,Z -71.212,A -90.000,B 90.000,C 0.000} C_DIS
LIN {X -38.814,Y -36.024,Z -70.611,A -90.000,B 90.000,C 0.000} C_DIS
LIN {X -38.626,Y -36.020,Z -70.455,A -90.000,B 90.000,C 0.000} C_DIS
LIN {X -38.407,Y -36.003,Z -70.278,A -90.000,B 90.000,C 0.000} C_DIS
LIN {X -38.049,Y -35.970,Z -69.991,A -90.000,B 90.000,C 0.000} C_DIS
LIN {X -37.716,Y -35.942,Z -69.745,A -90.000,B 90.000,C 0.000} C_DIS
LIN {X -37.570,Y -35.932,Z -69.646,A -90.000,B 90.000,C 0.000} C_DIS
LIN {X -37.240,Y -35.913,Z -69.437,A -90.000,B 90.000,C 0.000} C_DIS
LIN {X -37.014,Y -35.902,Z -69.309,A -90.000,B 90.000,C 0.000} C_DIS
LIN {X -36.760,Y -35.892,Z -69.180,A -90.000,B 90.000,C 0.000} C_DIS
LIN {X -36.375,Y -35.882,Z -69.003,A -90.000,B 90.000,C 0.000} C_DIS
LIN {X -36.146,Y -35.875,Z -68.902,A -90.000,B 90.000,C 0.000} C_DIS
LIN {X -35.879,Y -35.870,Z -68.795,A -90.000,B 90.000,C 0.000} C_DIS
LIN {X -35.646,Y -35.863,Z -68.704,A -90.000,B 90.000,C 0.000} C_DIS
LIN {X -35.379,Y -35.843,Z -68.604,A -90.000,B 90.000,C 0.000} C_DIS
LIN {X -34.764,Y -35.782,Z -68.380,A -90.000,B 90.000,C 0.000} C_DIS
LIN {X -34.561,Y -35.760,Z -68.309,A -90.000,B 90.000,C 0.000} C_DIS
LIN {X -34.370,Y -35.741,Z -68.249,A -90.000,B 90.000,C 0.000} C_DIS
LIN {X -34.288,Y -35.734,Z -68.226,A -90.000,B 90.000,C 0.000} C_DIS
LIN {X -33.588,Y -35.678,Z -68.039,A -90.000,B 90.000,C 0.000} C_DIS
LIN {X -33.129,Y -35.634,Z -67.920,A -90.000,B 90.000,C 0.000} C_DIS
LIN {X -32.885,Y -35.613,Z -67.864,A -90.000,B 90.000,C 0.000} C_DIS
LIN {X -32.506,Y -35.585,Z -67.786,A -90.000,B 90.000,C 0.000} C_DIS
LIN {X -31.958,Y -35.547,Z -67.680,A -90.000,B 90.000,C 0.000} C_DIS
LIN {X -31.744,Y -35.528,Z -67.649,A -90.000,B 90.000,C 0.000} C_DIS
LIN {X -31.580,Y -35.514,Z -67.628,A -90.000,B 90.000,C 0.000} C_DIS
LIN {X -31.483,Y -35.507,Z -67.618,A -90.000,B 90.000,C 0.000} C_DIS
LIN {X -30.852,Y -35.465,Z -67.568,A -90.000,B 90.000,C 0.000} C_DIS
LIN {X -30.723,Y -35.455,Z -67.559,A -90.000,B 90.000,C 0.000} C_DIS
LIN {X -29.949,Y -35.380,Z -67.511,A -90.000,B 90.000,C 0.000} C_DIS
LIN {X -29.726,Y -35.361,Z -67.503,A -90.000,B 90.000,C 0.000} C_DIS
LIN {X -29.323,Y -35.334,Z -67.505,A -90.000,B 90.000,C 0.000} C_DIS
LIN {X -29.037,Y -35.308,Z -67.517,A -90.000,B 90.000,C 0.000} C_DIS
LIN {X -29.037,Y -60.000,Z -67.517,A -90.000,B 90.000,C 0.000} C_DIS
LIN {X -45.901,Y -60.000,Z -76.595,A -90.000,B 90.000,C 0.000} C_DIS
LIN {X -45.901,Y -35.308,Z -76.595,A -90.000,B 90.000,C 0.000} C_DIS
LIN {X -45.849,Y -35.314,Z -76.491,A -90.000,B 90.000,C 0.000} C_DIS
LIN {X -45.665,Y -35.331,Z -76.142,A -90.000,B 90.000,C 0.000} C_DIS
LIN {X -45.547,Y -35.342,Z -75.929,A -90.000,B 90.000,C 0.000} C_DIS
LIN {X -45.287,Y -35.369,Z -75.488,A -90.000,B 90.000,C 0.000} C_DIS
LIN {X -45.097,Y -35.390,Z -75.188,A -90.000,B 90.000,C 0.000} C_DIS
LIN {X -44.285,Y -35.454,Z -73.923,A -90.000,B 90.000,C 0.000} C_DIS
LIN {X -44.154,Y -35.462,Z -73.723,A -90.000,B 90.000,C 0.000} C_DIS
LIN {X -43.767,Y -35.488,Z -73.168,A -90.000,B 90.000,C 0.000} C_DIS
LIN {X -43.419,Y -35.502,Z -72.675,A -90.000,B 90.000,C 0.000} C_DIS
LIN {X -43.218,Y -35.507,Z -72.394,A -90.000,B 90.000,C 0.000} C_DIS
LIN {X -42.974,Y -35.515,Z -72.081,A -90.000,B 90.000,C 0.000} C_DIS
LIN {X -42.457,Y -35.537,Z -71.461,A -90.000,B 90.000,C 0.000} C_DIS
LIN {X -42.169,Y -35.534,Z -71.125,A -90.000,B 90.000,C 0.000} C_DIS
LIN {X -41.995,Y -35.529,Z -70.930,A -90.000,B 90.000,C 0.000} C_DIS
LIN {X -41.774,Y -35.527,Z -70.698,A -90.000,B 90.000,C 0.000} C_DIS
LIN {X -41.154,Y -35.524,Z -70.078,A -90.000,B 90.000,C 0.000} C_DIS
LIN {X -40.912,Y -35.521,Z -69.853,A -90.000,B 90.000,C 0.000} C_DIS
LIN {X -40.746,Y -35.516,Z -69.708,A -90.000,B 90.000,C 0.000} C_DIS
LIN {X -39.788,Y -35.452,Z -68.927,A -90.000,B 90.000,C 0.000} C_DIS
LIN {X -39.262,Y -35.410,Z -68.503,A -90.000,B 90.000,C 0.000} C_DIS
LIN {X -38.916,Y -35.387,Z -68.244,A -90.000,B 90.000,C 0.000} C_DIS
LIN {X -38.793,Y -35.380,Z -68.155,A -90.000,B 90.000,C 0.000} C_DIS
LIN {X -38.584,Y -35.371,Z -68.016,A -90.000,B 90.000,C 0.000} C_DIS
LIN {X -38.408,Y -35.351,Z -67.907,A -90.000,B 90.000,C 0.000} C_DIS
LIN {X -38.268,Y -35.332,Z -67.823,A -90.000,B 90.000,C 0.000} C_DIS
LIN {X -38.065,Y -35.308,Z -67.712,A -90.000,B 90.000,C 0.000} C_DIS
LIN {X -38.065,Y -60.000,Z -67.712,A -90.000,B 90.000,C 0.000} C_DIS
LIN {X 13.661,Y -60.000,Z -172.527,A -90.000,B 90.000,C 0.000} C_DIS
LIN {X 13.661,Y -35.308,Z -172.527,A -90.000,B 90.000,C 0.000} C_DIS
LIN {X 13.947,Y -35.323,Z -172.232,A -90.000,B 90.000,C 0.000} C_DIS
LIN {X 14.038,Y -35.326,Z -172.132,A -90.000,B 90.000,C 0.000} C_DIS
LIN {X 15.025,Y -35.440,Z -170.988,A -90.000,B 90.000,C 0.000} C_DIS
LIN {X 15.502,Y -35.491,Z -170.436,A -90.000,B 90.000,C 0.000} C_DIS
LIN {X 15.733,Y -35.501,Z -170.152,A -90.000,B 90.000,C 0.000} C_DIS
LIN {X 16.266,Y -35.586,Z -169.452,A -90.000,B 90.000,C 0.000} C_DIS
LIN {X 16.397,Y -35.609,Z -169.276,A -90.000,B 90.000,C 0.000} C_DIS
LIN {X 17.098,Y -35.716,Z -168.230,A -90.000,B 90.000,C 0.000} C_DIS
LIN {X 17.497,Y -35.835,Z -167.596,A -90.000,B 90.000,C 0.000} C_DIS
LIN {X 18.053,Y -35.991,Z -166.628,A -90.000,B 90.000,C 0.000} C_DIS
LIN {X 18.143,Y -36.017,Z -166.471,A -90.000,B 90.000,C 0.000} C_DIS
LIN {X 18.271,Y -36.047,Z -166.178,A -90.000,B 90.000,C 0.000} C_DIS
LIN {X 18.314,Y -36.056,Z -166.083,A -90.000,B 90.000,C 0.000} C_DIS
LIN {X 18.420,Y -36.111,Z -165.845,A -90.000,B 90.000,C 0.000} C_DIS
LIN {X 18.702,Y -36.254,Z -165.267,A -90.000,B 90.000,C 0.000} C_DIS
LIN {X 18.706,Y -36.256,Z -165.256,A -90.000,B 90.000,C 0.000} C_DIS
LIN {X 18.627,Y -36.233,Z -165.155,A -90.000,B 90.000,C 0.000} C_DIS
LIN {X 18.540,Y -36.210,Z -165.032,A -90.000,B 90.000,C 0.000} C_DIS
LIN {X 18.431,Y -36.181,Z -164.865,A -90.000,B 90.000,C 0.000} C_DIS
LIN {X 18.360,Y -36.162,Z -164.748,A -90.000,B 90.000,C 0.000} C_DIS
LIN {X 18.243,Y -36.133,Z -164.539,A -90.000,B 90.000,C 0.000} C_DIS
LIN {X 18.173,Y -36.129,Z -164.419,A -90.000,B 90.000,C 0.000} C_DIS
LIN {X 18.110,Y -36.126,Z -164.302,A -90.000,B 90.000,C 0.000} C_DIS
LIN {X 18.075,Y -36.125,Z -164.234,A -90.000,B 90.000,C 0.000} C_DIS
LIN {X 17.860,Y -36.098,Z -163.963,A -90.000,B 90.000,C 0.000} C_DIS
LIN {X 17.742,Y -36.073,Z -163.808,A -90.000,B 90.000,C 0.000} C_DIS
LIN {X 17.665,Y -36.054,Z -163.702,A -90.000,B 90.000,C 0.000} C_DIS
LIN {X 17.598,Y -36.037,Z -163.603,A -90.000,B 90.000,C 0.000} C_DIS
LIN {X 17.556,Y -36.028,Z -163.537,A -90.000,B 90.000,C 0.000} C_DIS
LIN {X 17.258,Y -35.957,Z -163.066,A -90.000,B 90.000,C 0.000} C_DIS
LIN {X 17.132,Y -35.927,Z -162.835,A -90.000,B 90.000,C 0.000} C_DIS
LIN {X 17.080,Y -35.915,Z -162.731,A -90.000,B 90.000,C 0.000} C_DIS
LIN {X 16.954,Y -35.906,Z -162.487,A -90.000,B 90.000,C 0.000} C_DIS
LIN {X 16.897,Y -35.902,Z -162.371,A -90.000,B 90.000,C 0.000} C_DIS
LIN {X 16.836,Y -35.900,Z -162.239,A -90.000,B 90.000,C 0.000} C_DIS
LIN {X 16.631,Y -35.883,Z -161.846,A -90.000,B 90.000,C 0.000} C_DIS
LIN {X 16.501,Y -35.875,Z -161.570,A -90.000,B 90.000,C 0.000} C_DIS
LIN {X 16.409,Y -35.862,Z -161.367,A -90.000,B 90.000,C 0.000} C_DIS
LIN {X 16.210,Y -35.848,Z -160.937,A -90.000,B 90.000,C 0.000} C_DIS
LIN {X 16.112,Y -35.844,Z -160.710,A -90.000,B 90.000,C 0.000} C_DIS
LIN {X 16.002,Y -35.844,Z -160.415,A -90.000,B 90.000,C 0.000} C_DIS
LIN {X 15.888,Y -35.845,Z -160.064,A -90.000,B 90.000,C 0.000} C_DIS
LIN {X 15.835,Y -35.848,Z -159.890,A -90.000,B 90.000,C 0.000} C_DIS
LIN {X 15.505,Y -35.873,Z -158.749,A -90.000,B 90.000,C 0.000} C_DIS
LIN {X 15.384,Y -35.874,Z -158.370,A -90.000,B 90.000,C 0.000} C_DIS
LIN {X 15.337,Y -35.877,Z -158.220,A -90.000,B 90.000,C 0.000} C_DIS
LIN {X 15.279,Y -35.888,Z -157.999,A -90.000,B 90.000,C 0.000} C_DIS
LIN {X 15.242,Y -35.898,Z -157.835,A -90.000,B 90.000,C 0.000} C_DIS
LIN {X 15.093,Y -35.943,Z -157.145,A -90.000,B 90.000,C 0.000} C_DIS
LIN {X 15.046,Y -35.954,Z -156.908,A -90.000,B 90.000,C 0.000} C_DIS
LIN {X 14.992,Y -35.964,Z -156.565,A -90.000,B 90.000,C 0.000} C_DIS
LIN {X 14.950,Y -35.974,Z -156.246,A -90.000,B 90.000,C 0.000} C_DIS
LIN {X 14.863,Y -36.034,Z -155.675,A -90.000,B 90.000,C 0.000} C_DIS
LIN {X 14.825,Y -36.050,Z -155.397,A -90.000,B 90.000,C 0.000} C_DIS
LIN {X 14.775,Y -36.051,Z -154.983,A -90.000,B 90.000,C 0.000} C_DIS
LIN {X 14.760,Y -36.053,Z -154.811,A -90.000,B 90.000,C 0.000} C_DIS
LIN {X 14.752,Y -36.058,Z -154.613,A -90.000,B 90.000,C 0.000} C_DIS
LIN {X 14.753,Y -36.063,Z -154.486,A -90.000,B 90.000,C 0.000} C_DIS
LIN {X 14.757,Y -36.072,Z -154.284,A -90.000,B 90.000,C 0.000} C_DIS
LIN {X 14.588,Y -36.015,Z -154.313,A -90.000,B 90.000,C 0.000} C_DIS
LIN {X 14.259,Y -35.926,Z -154.358,A -90.000,B 90.000,C 0.000} C_DIS
LIN {X 14.053,Y -35.870,Z -154.382,A -90.000,B 90.000,C 0.000} C_DIS
LIN {X 13.519,Y -35.728,Z -154.435,A -90.000,B 90.000,C 0.000} C_DIS
LIN {X 13.299,Y -35.670,Z -154.452,A -90.000,B 90.000,C 0.000} C_DIS
LIN {X 12.743,Y -35.526,Z -154.481,A -90.000,B 90.000,C 0.000} C_DIS
LIN {X 12.072,Y -35.346,Z -154.554,A -90.000,B 90.000,C 0.000} C_DIS
LIN {X 11.930,Y -35.308,Z -154.569,A -90.000,B 90.000,C 0.000} C_DIS
LIN {X 11.878,Y -35.300,Z -154.577,A -90.000,B 90.000,C 0.000} C_DIS
LIN {X 11.733,Y -35.259,Z -154.605,A -90.000,B 90.000,C 0.000} C_DIS
LIN {X 11.647,Y -35.233,Z -154.631,A -90.000,B 90.000,C 0.000} C_DIS
LIN {X 11.570,Y -35.209,Z -154.661,A -90.000,B 90.000,C 0.000} C_DIS
LIN {X 11.500,Y -35.188,Z -154.696,A -90.000,B 90.000,C 0.000} C_DIS
LIN {X 11.439,Y -35.169,Z -154.736,A -90.000,B 90.000,C 0.000} C_DIS
LIN {X 11.384,Y -35.149,Z -154.780,A -90.000,B 90.000,C 0.000} C_DIS
LIN {X 11.338,Y -35.129,Z -154.828,A -90.000,B 90.000,C 0.000} C_DIS
LIN {X 11.298,Y -35.108,Z -154.880,A -90.000,B 90.000,C 0.000} C_DIS
LIN {X 11.264,Y -35.087,Z -154.934,A -90.000,B 90.000,C 0.000} C_DIS
LIN {X 11.237,Y -35.071,Z -154.993,A -90.000,B 90.000,C 0.000} C_DIS
LIN {X 11.210,Y -35.051,Z -155.088,A -90.000,B 90.000,C 0.000} C_DIS
LIN {X 11.199,Y -35.038,Z -155.154,A -90.000,B 90.000,C 0.000} C_DIS
LIN {X 11.193,Y -35.022,Z -155.258,A -90.000,B 90.000,C 0.000} C_DIS
LIN {X 11.196,Y -35.012,Z -155.330,A -90.000,B 90.000,C 0.000} C_DIS
LIN {X 11.211,Y -35.000,Z -155.442,A -90.000,B 90.000,C 0.000} C_DIS
LIN {X 11.236,Y -34.989,Z -155.558,A -90.000,B 90.000,C 0.000} C_DIS
LIN {X 11.286,Y -34.979,Z -155.716,A -90.000,B 90.000,C 0.000} C_DIS
LIN {X 11.351,Y -34.972,Z -155.877,A -90.000,B 90.000,C 0.000} C_DIS
LIN {X 11.430,Y -34.969,Z -156.038,A -90.000,B 90.000,C 0.000} C_DIS
LIN {X 11.522,Y -34.969,Z -156.199,A -90.000,B 90.000,C 0.000} C_DIS
LIN {X 11.624,Y -34.972,Z -156.358,A -90.000,B 90.000,C 0.000} C_DIS
LIN {X 11.735,Y -34.978,Z -156.511,A -90.000,B 90.000,C 0.000} C_DIS
LIN {X 11.793,Y -34.981,Z -156.585,A -90.000,B 90.000,C 0.000} C_DIS
LIN {X 11.913,Y -34.991,Z -156.728,A -90.000,B 90.000,C 0.000} C_DIS
LIN {X 11.974,Y -34.997,Z -156.796,A -90.000,B 90.000,C 0.000} C_DIS
LIN {X 12.099,Y -35.010,Z -156.924,A -90.000,B 90.000,C 0.000} C_DIS
LIN {X 12.225,Y -35.025,Z -157.039,A -90.000,B 90.000,C 0.000} C_DIS
LIN {X 12.349,Y -35.043,Z -157.140,A -90.000,B 90.000,C 0.000} C_DIS
LIN {X 12.471,Y -35.061,Z -157.225,A -90.000,B 90.000,C 0.000} C_DIS
LIN {X 12.588,Y -35.082,Z -157.292,A -90.000,B 90.000,C 0.000} C_DIS
LIN {X 12.644,Y -35.092,Z -157.318,A -90.000,B 90.000,C 0.000} C_DIS
LIN {X 12.698,Y -35.103,Z -157.338,A -90.000,B 90.000,C 0.000} C_DIS
LIN {X 12.750,Y -35.114,Z -157.353,A -90.000,B 90.000,C 0.000} C_DIS
LIN {X 12.800,Y -35.126,Z -157.363,A -90.000,B 90.000,C 0.000} C_DIS
LIN {X 12.847,Y -35.137,Z -157.366,A -90.000,B 90.000,C 0.000} C_DIS
LIN {X 12.891,Y -35.149,Z -157.364,A -90.000,B 90.000,C 0.000} C_DIS
LIN {X 12.933,Y -35.161,Z -157.354,A -90.000,B 90.000,C 0.000} C_DIS
LIN {X 12.970,Y -35.173,Z -157.339,A -90.000,B 90.000,C 0.000} C_DIS
LIN {X 13.020,Y -35.191,Z -157.302,A -90.000,B 90.000,C 0.000} C_DIS
LIN {X 13.049,Y -35.204,Z -157.268,A -90.000,B 90.000,C 0.000} C_DIS
LIN {X 13.073,Y -35.216,Z -157.227,A -90.000,B 90.000,C 0.000} C_DIS
LIN {X 13.101,Y -35.235,Z -157.150,A -90.000,B 90.000,C 0.000} C_DIS
LIN {X 13.119,Y -35.253,Z -157.056,A -90.000,B 90.000,C 0.000} C_DIS
LIN {X 13.125,Y -35.272,Z -156.942,A -90.000,B 90.000,C 0.000} C_DIS
LIN {X 13.117,Y -35.291,Z -156.808,A -90.000,B 90.000,C 0.000} C_DIS
LIN {X 13.099,Y -35.308,Z -156.654,A -90.000,B 90.000,C 0.000} C_DIS
LIN {X 13.067,Y -35.330,Z -156.452,A -90.000,B 90.000,C 0.000} C_DIS
LIN {X 13.001,Y -35.308,Z -156.454,A -90.000,B 90.000,C 0.000} C_DIS
LIN {X 13.001,Y -60.000,Z -156.454,A -90.000,B 90.000,C 0.000} C_DIS
LIN {X 16.233,Y -60.000,Z -165.984,A -90.000,B 90.000,C 0.000} C_DIS
LIN {X 16.233,Y -35.308,Z -165.984,A -90.000,B 90.000,C 0.000} C_DIS
LIN {X 16.283,Y -35.329,Z -165.893,A -90.000,B 90.000,C 0.000} C_DIS
LIN {X 16.470,Y -35.419,Z -165.546,A -90.000,B 90.000,C 0.000} C_DIS
LIN {X 16.543,Y -35.457,Z -165.363,A -90.000,B 90.000,C 0.000} C_DIS
LIN {X 16.508,Y -35.449,Z -165.294,A -90.000,B 90.000,C 0.000} C_DIS
LIN {X 16.280,Y -35.386,Z -164.988,A -90.000,B 90.000,C 0.000} C_DIS
LIN {X 16.213,Y -35.368,Z -164.895,A -90.000,B 90.000,C 0.000} C_DIS
LIN {X 16.064,Y -35.329,Z -164.673,A -90.000,B 90.000,C 0.000} C_DIS
LIN {X 15.997,Y -35.308,Z -164.564,A -90.000,B 90.000,C 0.000} C_DIS
LIN {X 15.997,Y -60.000,Z -164.564,A -90.000,B 90.000,C 0.000} C_DIS
LIN {X -92.570,Y -60.000,Z -243.561,A -90.000,B 90.000,C 0.000} C_DIS
LIN {X -92.570,Y -35.632,Z -243.561,A -90.000,B 90.000,C 0.000} C_DIS
LIN {X -92.552,Y -35.596,Z -243.498,A -90.000,B 90.000,C 0.000} C_DIS
LIN {X -92.516,Y -35.541,Z -243.394,A -90.000,B 90.000,C 0.000} C_DIS
LIN {X -92.371,Y -35.343,Z -243.012,A -90.000,B 90.000,C 0.000} C_DIS
LIN {X -92.344,Y -35.308,Z -242.943,A -90.000,B 90.000,C 0.000} C_DIS
LIN {X -92.329,Y -35.297,Z -242.903,A -90.000,B 90.000,C 0.000} C_DIS
LIN {X -92.317,Y -35.278,Z -242.867,A -90.000,B 90.000,C 0.000} C_DIS
LIN {X -92.309,Y -35.259,Z -242.835,A -90.000,B 90.000,C 0.000} C_DIS
LIN {X -92.302,Y -35.226,Z -242.783,A -90.000,B 90.000,C 0.000} C_DIS
LIN {X -92.303,Y -35.212,Z -242.763,A -90.000,B 90.000,C 0.000} C_DIS
LIN {X -92.314,Y -35.186,Z -242.734,A -90.000,B 90.000,C 0.000} C_DIS
LIN {X -92.324,Y -35.175,Z -242.725,A -90.000,B 90.000,C 0.000} C_DIS
LIN {X -92.336,Y -35.164,Z -242.719,A -90.000,B 90.000,C 0.000} C_DIS
LIN {X -92.350,Y -35.155,Z -242.716,A -90.000,B 90.000,C 0.000} C_DIS
LIN {X -92.367,Y -35.147,Z -242.716,A -90.000,B 90.000,C 0.000} C_DIS
LIN {X -92.407,Y -35.134,Z -242.725,A -90.000,B 90.000,C 0.000} C_DIS
LIN {X -92.454,Y -35.124,Z -242.744,A -90.000,B 90.000,C 0.000} C_DIS
LIN {X -92.508,Y -35.117,Z -242.772,A -90.000,B 90.000,C 0.000} C_DIS
LIN {X -92.567,Y -35.114,Z -242.809,A -90.000,B 90.000,C 0.000} C_DIS
LIN {X -92.631,Y -35.114,Z -242.853,A -90.000,B 90.000,C 0.000} C_DIS
LIN {X -92.699,Y -35.116,Z -242.903,A -90.000,B 90.000,C 0.000} C_DIS
LIN {X -92.840,Y -35.127,Z -243.017,A -90.000,B 90.000,C 0.000} C_DIS
LIN {X -92.912,Y -35.135,Z -243.079,A -90.000,B 90.000,C 0.000} C_DIS
LIN {X -93.053,Y -35.157,Z -243.209,A -90.000,B 90.000,C 0.000} C_DIS
LIN {X -93.121,Y -35.169,Z -243.273,A -90.000,B 90.000,C 0.000} C_DIS
LIN {X -93.244,Y -35.197,Z -243.398,A -90.000,B 90.000,C 0.000} C_DIS
LIN {X -93.344,Y -35.225,Z -243.509,A -90.000,B 90.000,C 0.000} C_DIS
LIN {X -93.384,Y -35.240,Z -243.557,A -90.000,B 90.000,C 0.000} C_DIS
LIN {X -93.427,Y -35.260,Z -243.616,A -90.000,B 90.000,C 0.000} C_DIS
LIN {X -93.447,Y -35.279,Z -243.656,A -90.000,B 90.000,C 0.000} C_DIS
LIN {X -93.446,Y -35.290,Z -243.671,A -90.000,B 90.000,C 0.000} C_DIS
LIN {X -93.440,Y -35.295,Z -243.674,A -90.000,B 90.000,C 0.000} C_DIS
LIN {X -93.432,Y -35.299,Z -243.675,A -90.000,B 90.000,C 0.000} C_DIS
LIN {X -93.405,Y -35.307,Z -243.667,A -90.000,B 90.000,C 0.000} C_DIS
LIN {X -93.385,Y -35.310,Z -243.658,A -90.000,B 90.000,C 0.000} C_DIS
LIN {X -93.336,Y -35.315,Z -243.631,A -90.000,B 90.000,C 0.000} C_DIS
LIN {X -93.305,Y -35.317,Z -243.611,A -90.000,B 90.000,C 0.000} C_DIS
LIN {X -93.230,Y -35.308,Z -243.561,A -90.000,B 90.000,C 0.000} C_DIS
LIN {X -90.775,Y -35.308,Z -241.848,A -90.000,B 90.000,C 0.000} C_DIS
LIN {X -88.791,Y -35.308,Z -240.483,A -90.000,B 90.000,C 0.000} C_DIS
LIN {X -87.689,Y -35.308,Z -239.729,A -90.000,B 90.000,C 0.000} C_DIS
LIN {X -87.545,Y -35.308,Z -239.633,A -90.000,B 90.000,C 0.000} C_DIS
LIN {X -83.935,Y -35.308,Z -237.310,A -90.000,B 90.000,C 0.000} C_DIS
LIN {X -82.894,Y -35.308,Z -236.645,A -90.000,B 90.000,C 0.000} C_DIS
LIN {X -79.632,Y -35.308,Z -234.574,A -90.000,B 90.000,C 0.000} C_DIS
LIN {X -79.428,Y -35.308,Z -234.449,A -90.000,B 90.000,C 0.000} C_DIS
LIN {X -77.531,Y -35.308,Z -233.329,A -90.000,B 90.000,C 0.000} C_DIS
LIN {X -71.021,Y -35.308,Z -229.514,A -90.000,B 90.000,C 0.000} C_DIS
LIN {X -67.382,Y -35.308,Z -227.563,A -90.000,B 90.000,C 0.000} C_DIS
LIN {X -62.414,Y -35.308,Z -224.961,A -90.000,B 90.000,C 0.000} C_DIS
LIN {X -62.146,Y -35.308,Z -224.824,A -90.000,B 90.000,C 0.000} C_DIS
LIN {X -59.254,Y -35.308,Z -223.374,A -90.000,B 90.000,C 0.000} C_DIS
LIN {X -53.658,Y -35.308,Z -220.594,A -90.000,B 90.000,C 0.000} C_DIS
LIN {X -46.050,Y -35.308,Z -216.843,A -90.000,B 90.000,C 0.000} C_DIS
LIN {X -45.792,Y -35.308,Z -216.717,A -90.000,B 90.000,C 0.000} C_DIS
LIN {X -45.391,Y -35.308,Z -216.517,A -90.000,B 90.000,C 0.000} C_DIS
LIN {X -38.905,Y -35.308,Z -213.307,A -90.000,B 90.000,C 0.000} C_DIS
LIN {X -36.159,Y -35.308,Z -211.881,A -90.000,B 90.000,C 0.000} C_DIS
LIN {X -33.374,Y -35.308,Z -210.396,A -90.000,B 90.000,C 0.000} C_DIS
LIN {X -32.019,Y -35.308,Z -209.641,A -90.000,B 90.000,C 0.000} C_DIS
LIN {X -28.550,Y -35.308,Z -207.672,A -90.000,B 90.000,C 0.000} C_DIS
LIN {X -28.308,Y -35.308,Z -207.525,A -90.000,B 90.000,C 0.000} C_DIS
LIN {X -27.289,Y -35.308,Z -206.901,A -90.000,B 90.000,C 0.000} C_DIS
LIN {X -24.897,Y -35.308,Z -205.466,A -90.000,B 90.000,C 0.000} C_DIS
LIN {X -24.345,Y -35.308,Z -205.130,A -90.000,B 90.000,C 0.000} C_DIS
LIN {X -21.650,Y -35.308,Z -203.363,A -90.000,B 90.000,C 0.000} C_DIS
LIN {X -20.725,Y -35.308,Z -202.746,A -90.000,B 90.000,C 0.000} C_DIS
LIN {X -19.325,Y -35.308,Z -201.730,A -90.000,B 90.000,C 0.000} C_DIS
LIN {X -17.267,Y -35.308,Z -200.258,A -90.000,B 90.000,C 0.000} C_DIS
LIN {X -15.473,Y -35.308,Z -198.859,A -90.000,B 90.000,C 0.000} C_DIS
LIN {X -13.776,Y -35.308,Z -197.557,A -90.000,B 90.000,C 0.000} C_DIS
LIN {X -11.730,Y -35.308,Z -195.876,A -90.000,B 90.000,C 0.000} C_DIS
LIN {X -10.294,Y -35.308,Z -194.714,A -90.000,B 90.000,C 0.000} C_DIS
LIN {X -7.946,Y -35.308,Z -192.722,A -90.000,B 90.000,C 0.000} C_DIS
LIN {X -6.719,Y -35.308,Z -191.694,A -90.000,B 90.000,C 0.000} C_DIS
LIN {X -5.606,Y -35.308,Z -190.747,A -90.000,B 90.000,C 0.000} C_DIS
LIN {X -2.954,Y -35.308,Z -188.461,A -90.000,B 90.000,C 0.000} C_DIS
LIN {X -2.200,Y -35.308,Z -187.804,A -90.000,B 90.000,C 0.000} C_DIS
LIN {X 0.816,Y -35.308,Z -185.158,A -90.000,B 90.000,C 0.000} C_DIS
LIN {X 4.247,Y -35.308,Z -182.081,A -90.000,B 90.000,C 0.000} C_DIS
LIN {X 7.403,Y -35.308,Z -179.171,A -90.000,B 90.000,C 0.000} C_DIS
LIN {X 7.987,Y -35.308,Z -178.599,A -90.000,B 90.000,C 0.000} C_DIS
LIN {X 9.969,Y -35.308,Z -176.679,A -90.000,B 90.000,C 0.000} C_DIS
LIN {X 10.479,Y -35.308,Z -176.113,A -90.000,B 90.000,C 0.000} C_DIS
LIN {X 12.241,Y -35.308,Z -174.268,A -90.000,B 90.000,C 0.000} C_DIS
LIN {X 12.936,Y -35.308,Z -173.380,A -90.000,B 90.000,C 0.000} C_DIS
LIN {X 14.011,Y -35.308,Z -172.116,A -90.000,B 90.000,C 0.000} C_DIS
LIN {X 15.038,Y -35.308,Z -170.522,A -90.000,B 90.000,C 0.000} C_DIS
LIN {X 15.242,Y -35.308,Z -170.211,A -90.000,B 90.000,C 0.000} C_DIS
LIN {X 15.295,Y -35.308,Z -170.122,A -90.000,B 90.000,C 0.000} C_DIS
LIN {X 15.572,Y -35.308,Z -169.342,A -90.000,B 90.000,C 0.000} C_DIS
LIN {X 16.191,Y -35.308,Z -167.696,A -90.000,B 90.000,C 0.000} C_DIS
LIN {X 16.202,Y -35.308,Z -166.977,A -90.000,B 90.000,C 0.000} C_DIS
LIN {X 16.235,Y -35.308,Z -165.941,A -90.000,B 90.000,C 0.000} C_DIS
LIN {X 16.027,Y -35.308,Z -164.783,A -90.000,B 90.000,C 0.000} C_DIS
LIN {X 15.997,Y -35.308,Z -164.567,A -90.000,B 90.000,C 0.000} C_DIS
LIN {X 15.950,Y -35.308,Z -164.190,A -90.000,B 90.000,C 0.000} C_DIS
LIN {X 15.688,Y -35.308,Z -163.046,A -90.000,B 90.000,C 0.000} C_DIS
LIN {X 15.580,Y -35.308,Z -162.786,A -90.000,B 90.000,C 0.000} C_DIS
LIN {X 15.477,Y -35.308,Z -162.527,A -90.000,B 90.000,C 0.000} C_DIS
LIN {X 15.213,Y -35.308,Z -161.611,A -90.000,B 90.000,C 0.000} C_DIS
LIN {X 14.879,Y -35.308,Z -160.748,A -90.000,B 90.000,C 0.000} C_DIS
LIN {X 14.668,Y -35.308,Z -160.176,A -90.000,B 90.000,C 0.000} C_DIS
LIN {X 14.296,Y -35.308,Z -159.239,A -90.000,B 90.000,C 0.000} C_DIS
LIN {X 14.181,Y -35.308,Z -159.016,A -90.000,B 90.000,C 0.000} C_DIS
LIN {X 13.717,Y -35.308,Z -157.939,A -90.000,B 90.000,C 0.000} C_DIS
LIN {X 13.557,Y -35.308,Z -157.551,A -90.000,B 90.000,C 0.000} C_DIS
LIN {X 13.535,Y -35.308,Z -157.519,A -90.000,B 90.000,C 0.000} C_DIS
LIN {X 13.403,Y -35.308,Z -157.271,A -90.000,B 90.000,C 0.000} C_DIS
LIN {X 13.001,Y -35.308,Z -156.454,A -90.000,B 90.000,C 0.000} C_DIS
LIN {X 12.675,Y -35.308,Z -155.759,A -90.000,B 90.000,C 0.000} C_DIS
LIN {X 12.631,Y -35.308,Z -155.624,A -90.000,B 90.000,C 0.000} C_DIS
LIN {X 11.889,Y -35.308,Z -154.505,A -90.000,B 90.000,C 0.000} C_DIS
LIN {X 11.779,Y -35.308,Z -154.327,A -90.000,B 90.000,C 0.000} C_DIS
LIN {X 10.772,Y -35.308,Z -153.591,A -90.000,B 90.000,C 0.000} C_DIS
LIN {X 9.480,Y -35.308,Z -153.395,A -90.000,B 90.000,C 0.000} C_DIS
LIN {X 9.181,Y -35.308,Z -153.407,A -90.000,B 90.000,C 0.000} C_DIS
LIN {X 8.520,Y -35.308,Z -153.486,A -90.000,B 90.000,C 0.000} C_DIS
LIN {X 7.164,Y -35.308,Z -153.674,A -90.000,B 90.000,C 0.000} C_DIS
LIN {X 6.741,Y -35.308,Z -153.703,A -90.000,B 90.000,C 0.000} C_DIS
LIN {X 5.739,Y -35.308,Z -153.708,A -90.000,B 90.000,C 0.000} C_DIS
LIN {X 3.891,Y -35.308,Z -153.770,A -90.000,B 90.000,C 0.000} C_DIS
LIN {X 3.464,Y -35.308,Z -153.766,A -90.000,B 90.000,C 0.000} C_DIS
LIN {X 3.451,Y -35.308,Z -153.765,A -90.000,B 90.000,C 0.000} C_DIS
LIN {X 3.170,Y -35.308,Z -153.735,A -90.000,B 90.000,C 0.000} C_DIS
LIN {X 0.424,Y -35.308,Z -153.516,A -90.000,B 90.000,C 0.000} C_DIS
LIN {X 0.304,Y -35.308,Z -153.502,A -90.000,B 90.000,C 0.000} C_DIS
LIN {X 0.230,Y -35.308,Z -153.497,A -90.000,B 90.000,C 0.000} C_DIS
LIN {X 0.117,Y -35.308,Z -153.479,A -90.000,B 90.000,C 0.000} C_DIS
LIN {X -0.017,Y -35.308,Z -153.462,A -90.000,B 90.000,C 0.000} C_DIS
LIN {X -0.089,Y -35.308,Z -153.446,A -90.000,B 90.000,C 0.000} C_DIS
LIN {X -0.219,Y -35.308,Z -153.426,A -90.000,B 90.000,C 0.000} C_DIS
LIN {X -3.276,Y -35.308,Z -152.828,A -90.000,B 90.000,C 0.000} C_DIS
LIN {X -3.533,Y -35.308,Z -152.781,A -90.000,B 90.000,C 0.000} C_DIS
LIN {X -3.973,Y -35.308,Z -152.661,A -90.000,B 90.000,C 0.000} C_DIS
LIN {X -6.124,Y -35.308,Z -152.010,A -90.000,B 90.000,C 0.000} C_DIS
LIN {X -7.476,Y -35.308,Z -151.597,A -90.000,B 90.000,C 0.000} C_DIS
LIN {X -7.901,Y -35.308,Z -151.429,A -90.000,B 90.000,C 0.000} C_DIS
LIN {X -11.490,Y -35.308,Z -149.963,A -90.000,B 90.000,C 0.000} C_DIS
LIN {X -13.616,Y -35.308,Z -148.851,A -90.000,B 90.000,C 0.000} C_DIS
LIN {X -15.410,Y -35.308,Z -147.915,A -90.000,B 90.000,C 0.000} C_DIS
LIN {X -15.601,Y -35.308,Z -147.814,A -90.000,B 90.000,C 0.000} C_DIS
LIN {X -16.756,Y -35.308,Z -147.058,A -90.000,B 90.000,C 0.000} C_DIS
LIN {X -19.225,Y -35.308,Z -145.469,A -90.000,B 90.000,C 0.000} C_DIS
LIN {X -19.612,Y -35.308,Z -145.209,A -90.000,B 90.000,C 0.000} C_DIS
LIN {X -22.240,Y -35.308,Z -143.140,A -90.000,B 90.000,C 0.000} C_DIS
LIN {X -23.092,Y -35.308,Z -142.478,A -90.000,B 90.000,C 0.000} C_DIS
LIN {X -23.450,Y -35.308,Z -142.177,A -90.000,B 90.000,C 0.000} C_DIS
LIN {X -24.062,Y -35.308,Z -141.610,A -90.000,B 90.000,C 0.000} C_DIS
LIN {X -24.924,Y -35.308,Z -140.828,A -90.000,B 90.000,C 0.000} C_DIS
LIN {X -26.582,Y -35.308,Z -139.293,A -90.000,B 90.000,C 0.000} C_DIS
LIN {X -26.896,Y -35.308,Z -138.961,A -90.000,B 90.000,C 0.000} C_DIS
LIN {X -27.184,Y -35.308,Z -138.641,A -90.000,B 90.000,C 0.000} C_DIS
LIN {X -28.692,Y -35.308,Z -136.954,A -90.000,B 90.000,C 0.000} C_DIS
LIN {X -29.617,Y -35.308,Z -135.924,A -90.000,B 90.000,C 0.000} C_DIS
LIN {X -29.891,Y -35.308,Z -135.560,A -90.000,B 90.000,C 0.000} C_DIS
LIN {X -31.804,Y -35.308,Z -132.936,A -90.000,B 90.000,C 0.000} C_DIS
LIN {X -32.082,Y -35.308,Z -132.540,A -90.000,B 90.000,C 0.000} C_DIS
LIN {X -32.314,Y -35.308,Z -132.150,A -90.000,B 90.000,C 0.000} C_DIS
LIN {X -33.818,Y -35.308,Z -129.500,A -90.000,B 90.000,C 0.000} C_DIS
LIN {X -34.003,Y -35.308,Z -129.166,A -90.000,B 90.000,C 0.000} C_DIS
LIN {X -34.250,Y -35.308,Z -128.626,A -90.000,B 90.000,C 0.000} C_DIS
LIN {X -35.514,Y -35.308,Z -125.817,A -90.000,B 90.000,C 0.000} C_DIS
LIN {X -35.728,Y -35.308,Z -125.222,A -90.000,B 90.000,C 0.000} C_DIS
LIN {X -36.551,Y -35.308,Z -122.960,A -90.000,B 90.000,C 0.000} C_DIS
LIN {X -36.688,Y -35.308,Z -122.541,A -90.000,B 90.000,C 0.000} C_DIS
LIN {X -36.770,Y -35.308,Z -122.250,A -90.000,B 90.000,C 0.000} C_DIS
LIN {X -37.212,Y -35.308,Z -120.772,A -90.000,B 90.000,C 0.000} C_DIS
LIN {X -37.513,Y -35.308,Z -119.701,A -90.000,B 90.000,C 0.000} C_DIS
LIN {X -37.615,Y -35.308,Z -119.213,A -90.000,B 90.000,C 0.000} C_DIS
LIN {X -37.917,Y -35.308,Z -117.679,A -90.000,B 90.000,C 0.000} C_DIS
LIN {X -38.177,Y -35.308,Z -116.454,A -90.000,B 90.000,C 0.000} C_DIS
LIN {X -38.232,Y -35.308,Z -116.187,A -90.000,B 90.000,C 0.000} C_DIS
LIN {X -38.317,Y -35.308,Z -115.491,A -90.000,B 90.000,C 0.000} C_DIS
LIN {X -38.490,Y -35.308,Z -114.301,A -90.000,B 90.000,C 0.000} C_DIS
LIN {X -38.614,Y -35.308,Z -113.241,A -90.000,B 90.000,C 0.000} C_DIS
LIN {X -38.656,Y -35.308,Z -112.793,A -90.000,B 90.000,C 0.000} C_DIS
LIN {X -38.664,Y -35.308,Z -112.598,A -90.000,B 90.000,C 0.000} C_DIS
LIN {X -38.691,Y -35.308,Z -111.240,A -90.000,B 90.000,C 0.000} C_DIS
LIN {X -38.753,Y -35.308,Z -109.527,A -90.000,B 90.000,C 0.000} C_DIS
LIN {X -38.743,Y -35.308,Z -109.086,A -90.000,B 90.000,C 0.000} C_DIS
LIN {X -38.716,Y -35.308,Z -108.698,A -90.000,B 90.000,C 0.000} C_DIS
LIN {X -38.508,Y -35.308,Z -106.379,A -90.000,B 90.000,C 0.000} C_DIS
LIN {X -38.481,Y -35.308,Z -106.177,A -90.000,B 90.000,C 0.000} C_DIS
LIN {X -38.448,Y -35.308,Z -105.942,A -90.000,B 90.000,C 0.000} C_DIS
LIN {X -38.109,Y -35.308,Z -104.075,A -90.000,B 90.000,C 0.000} C_DIS
LIN {X -38.014,Y -35.308,Z -103.537,A -90.000,B 90.000,C 0.000} C_DIS
LIN {X -37.765,Y -35.308,Z -102.500,A -90.000,B 90.000,C 0.000} C_DIS
LIN {X -37.732,Y -35.308,Z -102.310,A -90.000,B 90.000,C 0.000} C_DIS
LIN {X -37.753,Y -35.308,Z -102.246,A -90.000,B 90.000,C 0.000} C_DIS
LIN {X -38.049,Y -35.308,Z -101.780,A -90.000,B 90.000,C 0.000} C_DIS
LIN {X -38.273,Y -35.308,Z -101.417,A -90.000,B 90.000,C 0.000} C_DIS
LIN {X -38.812,Y -35.308,Z -100.710,A -90.000,B 90.000,C 0.000} C_DIS
LIN {X -39.424,Y -35.308,Z -99.884,A -90.000,B 90.000,C 0.000} C_DIS
LIN {X -40.029,Y -35.308,Z -99.020,A -90.000,B 90.000,C 0.000} C_DIS
LIN {X -40.466,Y -35.308,Z -98.394,A -90.000,B 90.000,C 0.000} C_DIS
LIN {X -40.645,Y -35.308,Z -98.130,A -90.000,B 90.000,C 0.000} C_DIS
LIN {X -41.583,Y -35.308,Z -96.608,A -90.000,B 90.000,C 0.000} C_DIS
LIN {X -42.164,Y -35.308,Z -95.640,A -90.000,B 90.000,C 0.000} C_DIS
LIN {X -42.494,Y -35.308,Z -95.046,A -90.000,B 90.000,C 0.000} C_DIS
LIN {X -42.673,Y -35.308,Z -94.710,A -90.000,B 90.000,C 0.000} C_DIS
LIN {X -43.408,Y -35.308,Z -93.348,A -90.000,B 90.000,C 0.000} C_DIS
LIN {X -43.996,Y -35.308,Z -92.203,A -90.000,B 90.000,C 0.000} C_DIS
LIN {X -44.233,Y -35.308,Z -91.694,A -90.000,B 90.000,C 0.000} C_DIS
LIN {X -44.945,Y -35.308,Z -90.007,A -90.000,B 90.000,C 0.000} C_DIS
LIN {X -45.074,Y -35.308,Z -89.692,A -90.000,B 90.000,C 0.000} C_DIS
LIN {X -45.342,Y -35.308,Z -88.992,A -90.000,B 90.000,C 0.000} C_DIS
LIN {X -45.558,Y -35.308,Z -88.419,A -90.000,B 90.000,C 0.000} C_DIS
LIN {X -45.729,Y -35.308,Z -87.882,A -90.000,B 90.000,C 0.000} C_DIS
LIN {X -45.932,Y -35.308,Z -87.146,A -90.000,B 90.000,C 0.000} C_DIS
LIN {X -46.432,Y -35.308,Z -85.011,A -90.000,B 90.000,C 0.000} C_DIS
LIN {X -46.516,Y -35.308,Z -84.667,A -90.000,B 90.000,C 0.000} C_DIS
LIN {X -46.554,Y -35.308,Z -84.388,A -90.000,B 90.000,C 0.000} C_DIS
LIN {X -46.593,Y -35.308,Z -84.067,A -90.000,B 90.000,C 0.000} C_DIS
LIN {X -46.770,Y -35.308,Z -82.248,A -90.000,B 90.000,C 0.000} C_DIS
LIN {X -46.731,Y -35.308,Z -81.380,A -90.000,B 90.000,C 0.000} C_DIS
LIN {X -46.726,Y -35.308,Z -81.257,A -90.000,B 90.000,C 0.000} C_DIS
LIN {X -46.656,Y -35.308,Z -80.059,A -90.000,B 90.000,C 0.000} C_DIS
LIN {X -46.494,Y -35.308,Z -79.067,A -90.000,B 90.000,C 0.000} C_DIS
LIN {X -46.376,Y -35.308,Z -78.468,A -90.000,B 90.000,C 0.000} C_DIS
LIN {X -46.282,Y -35.308,Z -78.009,A -90.000,B 90.000,C 0.000} C_DIS
LIN {X -45.931,Y -35.308,Z -76.696,A -90.000,B 90.000,C 0.000} C_DIS
LIN {X -45.862,Y -35.308,Z -76.469,A -90.000,B 90.000,C 0.000} C_DIS
LIN {X -45.738,Y -35.308,Z -76.099,A -90.000,B 90.000,C 0.000} C_DIS
LIN {X -45.303,Y -35.308,Z -74.880,A -90.000,B 90.000,C 0.000} C_DIS
LIN {X -45.124,Y -35.308,Z -74.471,A -90.000,B 90.000,C 0.000} C_DIS
LIN {X -44.663,Y -35.308,Z -73.394,A -90.000,B 90.000,C 0.000} C_DIS
LIN {X -44.405,Y -35.308,Z -72.869,A -90.000,B 90.000,C 0.000} C_DIS
LIN {X -44.290,Y -35.308,Z -72.662,A -90.000,B 90.000,C 0.000} C_DIS
LIN {X -43.796,Y -35.308,Z -71.839,A -90.000,B 90.000,C 0.000} C_DIS
LIN {X -43.337,Y -35.308,Z -71.144,A -90.000,B 90.000,C 0.000} C_DIS
LIN {X -43.181,Y -35.308,Z -70.966,A -90.000,B 90.000,C 0.000} C_DIS
LIN {X -42.729,Y -35.308,Z -70.482,A -90.000,B 90.000,C 0.000} C_DIS
LIN {X -41.818,Y -35.308,Z -69.575,A -90.000,B 90.000,C 0.000} C_DIS
LIN {X -41.628,Y -35.308,Z -69.433,A -90.000,B 90.000,C 0.000} C_DIS
LIN {X -41.395,Y -35.308,Z -69.276,A -90.000,B 90.000,C 0.000} C_DIS
LIN {X -40.111,Y -35.308,Z -68.557,A -90.000,B 90.000,C 0.000} C_DIS
LIN {X -38.875,Y -35.308,Z -67.930,A -90.000,B 90.000,C 0.000} C_DIS
LIN {X -38.604,Y -35.308,Z -67.849,A -90.000,B 90.000,C 0.000} C_DIS
LIN {X -37.617,Y -35.308,Z -67.597,A -90.000,B 90.000,C 0.000} C_DIS
LIN {X -36.469,Y -35.308,Z -67.400,A -90.000,B 90.000,C 0.000} C_DIS
LIN {X -34.698,Y -35.308,Z -67.179,A -90.000,B 90.000,C 0.000} C_DIS
LIN {X -34.425,Y -35.308,Z -67.148,A -90.000,B 90.000,C 0.000} C_DIS
LIN {X -34.379,Y -35.308,Z -67.145,A -90.000,B 90.000,C 0.000} C_DIS
LIN {X -32.616,Y -35.308,Z -67.116,A -90.000,B 90.000,C 0.000} C_DIS
LIN {X -32.073,Y -35.308,Z -67.136,A -90.000,B 90.000,C 0.000} C_DIS
LIN {X -31.551,Y -35.308,Z -67.180,A -90.000,B 90.000,C 0.000} C_DIS
LIN {X -29.822,Y -35.308,Z -67.391,A -90.000,B 90.000,C 0.000} C_DIS
LIN {X -29.369,Y -35.308,Z -67.452,A -90.000,B 90.000,C 0.000} C_DIS
LIN {X -29.297,Y -35.308,Z -67.463,A -90.000,B 90.000,C 0.000} C_DIS
LIN {X -27.472,Y -35.308,Z -67.842,A -90.000,B 90.000,C 0.000} C_DIS
LIN {X -27.129,Y -35.308,Z -67.918,A -90.000,B 90.000,C 0.000} C_DIS
LIN {X -26.855,Y -35.308,Z -67.983,A -90.000,B 90.000,C 0.000} C_DIS
LIN {X -25.302,Y -35.308,Z -68.446,A -90.000,B 90.000,C 0.000} C_DIS
LIN {X -25.009,Y -35.308,Z -68.540,A -90.000,B 90.000,C 0.000} C_DIS
LIN {X -23.648,Y -35.308,Z -68.995,A -90.000,B 90.000,C 0.000} C_DIS
LIN {X -23.389,Y -35.308,Z -69.087,A -90.000,B 90.000,C 0.000} C_DIS
LIN {X -22.243,Y -35.308,Z -69.426,A -90.000,B 90.000,C 0.000} C_DIS
LIN {X -22.128,Y -35.308,Z -69.462,A -90.000,B 90.000,C 0.000} C_DIS
LIN {X -21.489,Y -35.308,Z -69.558,A -90.000,B 90.000,C 0.000} C_DIS
LIN {X -21.182,Y -35.308,Z -69.503,A -90.000,B 90.000,C 0.000} C_DIS
LIN {X -21.007,Y -35.308,Z -69.432,A -90.000,B 90.000,C 0.000} C_DIS
LIN {X -20.638,Y -35.308,Z -69.286,A -90.000,B 90.000,C 0.000} C_DIS
LIN {X -20.154,Y -35.308,Z -69.081,A -90.000,B 90.000,C 0.000} C_DIS
LIN {X -19.466,Y -35.308,Z -68.808,A -90.000,B 90.000,C 0.000} C_DIS
LIN {X -19.109,Y -35.308,Z -68.681,A -90.000,B 90.000,C 0.000} C_DIS
LIN {X -17.798,Y -35.308,Z -68.354,A -90.000,B 90.000,C 0.000} C_DIS
LIN {X -17.298,Y -35.308,Z -68.201,A -90.000,B 90.000,C 0.000} C_DIS
LIN {X -16.954,Y -35.308,Z -68.129,A -90.000,B 90.000,C 0.000} C_DIS
LIN {X -15.815,Y -35.308,Z -67.987,A -90.000,B 90.000,C 0.000} C_DIS
LIN {X -14.927,Y -35.308,Z -67.901,A -90.000,B 90.000,C 0.000} C_DIS
LIN {X -14.214,Y -35.308,Z -67.719,A -90.000,B 90.000,C 0.000} C_DIS
LIN {X -13.928,Y -35.308,Z -67.686,A -90.000,B 90.000,C 0.000} C_DIS
LIN {X -13.730,Y -35.308,Z -67.667,A -90.000,B 90.000,C 0.000} C_DIS
LIN {X -12.932,Y -35.308,Z -67.408,A -90.000,B 90.000,C 0.000} C_DIS
LIN {X -12.669,Y -35.308,Z -67.178,A -90.000,B 90.000,C 0.000} C_DIS
LIN {X -12.224,Y -35.308,Z -66.741,A -90.000,B 90.000,C 0.000} C_DIS
LIN {X -11.890,Y -35.308,Z -66.381,A -90.000,B 90.000,C 0.000} C_DIS
LIN {X -11.628,Y -35.308,Z -66.089,A -90.000,B 90.000,C 0.000} C_DIS
LIN {X -11.502,Y -35.308,Z -65.961,A -90.000,B 90.000,C 0.000} C_DIS
LIN {X -11.346,Y -35.308,Z -65.873,A -90.000,B 90.000,C 0.000} C_DIS
LIN {X -10.449,Y -35.308,Z -65.624,A -90.000,B 90.000,C 0.000} C_DIS
LIN {X -10.232,Y -35.308,Z -65.574,A -90.000,B 90.000,C 0.000} C_DIS
LIN {X -10.001,Y -35.308,Z -65.522,A -90.000,B 90.000,C 0.000} C_DIS
LIN {X -8.447,Y -35.308,Z -65.275,A -90.000,B 90.000,C 0.000} C_DIS
LIN {X -6.606,Y -35.308,Z -65.227,A -90.000,B 90.000,C 0.000} C_DIS
LIN {X -5.922,Y -35.308,Z -65.245,A -90.000,B 90.000,C 0.000} C_DIS
LIN {X -3.800,Y -35.308,Z -65.248,A -90.000,B 90.000,C 0.000} C_DIS
LIN {X -1.928,Y -35.308,Z -65.308,A -90.000,B 90.000,C 0.000} C_DIS
LIN {X -1.873,Y -35.308,Z -65.305,A -90.000,B 90.000,C 0.000} C_DIS
LIN {X 1.007,Y -35.308,Z -65.299,A -90.000,B 90.000,C 0.000} C_DIS
LIN {X 1.568,Y -35.308,Z -65.305,A -90.000,B 90.000,C 0.000} C_DIS
LIN {X 2.404,Y -35.308,Z -65.277,A -90.000,B 90.000,C 0.000} C_DIS
LIN {X 4.482,Y -35.308,Z -65.277,A -90.000,B 90.000,C 0.000} C_DIS
LIN {X 5.941,Y -35.308,Z -65.199,A -90.000,B 90.000,C 0.000} C_DIS
LIN {X 6.808,Y -35.308,Z -65.186,A -90.000,B 90.000,C 0.000} C_DIS
LIN {X 7.534,Y -35.308,Z -65.184,A -90.000,B 90.000,C 0.000} C_DIS
LIN {X 8.767,Y -35.308,Z -65.221,A -90.000,B 90.000,C 0.000} C_DIS
LIN {X 9.124,Y -35.308,Z -65.229,A -90.000,B 90.000,C 0.000} C_DIS
LIN {X 9.502,Y -35.308,Z -65.250,A -90.000,B 90.000,C 0.000} C_DIS
LIN {X 10.460,Y -35.308,Z -65.325,A -90.000,B 90.000,C 0.000} C_DIS
LIN {X 10.701,Y -35.308,Z -65.327,A -90.000,B 90.000,C 0.000} C_DIS
LIN {X 11.096,Y -35.308,Z -65.350,A -90.000,B 90.000,C 0.000} C_DIS
LIN {X 11.638,Y -35.308,Z -65.403,A -90.000,B 90.000,C 0.000} C_DIS
LIN {X 12.084,Y -35.308,Z -65.375,A -90.000,B 90.000,C 0.000} C_DIS
LIN {X 12.233,Y -35.308,Z -65.379,A -90.000,B 90.000,C 0.000} C_DIS
LIN {X 12.285,Y -35.308,Z -65.364,A -90.000,B 90.000,C 0.000} C_DIS
LIN {X 12.399,Y -35.308,Z -65.251,A -90.000,B 90.000,C 0.000} C_DIS
LIN {X 12.619,Y -35.308,Z -64.991,A -90.000,B 90.000,C 0.000} C_DIS
LIN {X 13.177,Y -35.308,Z -64.476,A -90.000,B 90.000,C 0.000} C_DIS
LIN {X 13.458,Y -35.308,Z -64.221,A -90.000,B 90.000,C 0.000} C_DIS
LIN {X 13.775,Y -35.308,Z -64.003,A -90.000,B 90.000,C 0.000} C_DIS
LIN {X 14.675,Y -35.308,Z -63.539,A -90.000,B 90.000,C 0.000} C_DIS
LIN {X 15.041,Y -35.308,Z -63.408,A -90.000,B 90.000,C 0.000} C_DIS
LIN {X 15.201,Y -35.308,Z -63.370,A -90.000,B 90.000,C 0.000} C_DIS
LIN {X 15.420,Y -35.308,Z -63.324,A -90.000,B 90.000,C 0.000} C_DIS
LIN {X 15.584,Y -35.308,Z -63.307,A -90.000,B 90.000,C 0.000} C_DIS
LIN {X 16.223,Y -35.308,Z -63.250,A -90.000,B 90.000,C 0.000} C_DIS
LIN {X 16.482,Y -35.308,Z -63.230,A -90.000,B 90.000,C 0.000} C_DIS
LIN {X 16.885,Y -35.308,Z -63.241,A -90.000,B 90.000,C 0.000} C_DIS
LIN {X 17.580,Y -35.308,Z -63.333,A -90.000,B 90.000,C 0.000} C_DIS
LIN {X 17.979,Y -35.308,Z -63.391,A -90.000,B 90.000,C 0.000} C_DIS
LIN {X 18.145,Y -35.308,Z -63.431,A -90.000,B 90.000,C 0.000} C_DIS
LIN {X 18.238,Y -35.308,Z -63.381,A -90.000,B 90.000,C 0.000} C_DIS
LIN {X 18.398,Y -35.308,Z -63.199,A -90.000,B 90.000,C 0.000} C_DIS
LIN {X 18.704,Y -35.308,Z -62.927,A -90.000,B 90.000,C 0.000} C_DIS
LIN {X 18.749,Y -35.308,Z -62.892,A -90.000,B 90.000,C 0.000} C_DIS
LIN {X 19.192,Y -35.308,Z -62.589,A -90.000,B 90.000,C 0.000} C_DIS
LIN {X 19.215,Y -35.308,Z -62.574,A -90.000,B 90.000,C 0.000} C_DIS
LIN {X 19.573,Y -35.308,Z -62.389,A -90.000,B 90.000,C 0.000} C_DIS
LIN {X 19.951,Y -35.308,Z -62.250,A -90.000,B 90.000,C 0.000} C_DIS
LIN {X 20.343,Y -35.308,Z -62.159,A -90.000,B 90.000,C 0.000} C_DIS
LIN {X 20.744,Y -35.308,Z -62.117,A -90.000,B 90.000,C 0.000} C_DIS
LIN {X 21.147,Y -35.308,Z -62.125,A -90.000,B 90.000,C 0.000} C_DIS
LIN {X 21.177,Y -35.308,Z -62.129,A -90.000,B 90.000,C 0.000} C_DIS
LIN {X 21.299,Y -35.308,Z -62.131,A -90.000,B 90.000,C 0.000} C_DIS
LIN {X 21.698,Y -35.308,Z -62.189,A -90.000,B 90.000,C 0.000} C_DIS
LIN {X 21.882,Y -35.308,Z -62.229,A -90.000,B 90.000,C 0.000} C_DIS
LIN {X 22.104,Y -35.308,Z -62.289,A -90.000,B 90.000,C 0.000} C_DIS
LIN {X 22.505,Y -35.308,Z -62.426,A -90.000,B 90.000,C 0.000} C_DIS
LIN {X 22.548,Y -35.308,Z -62.447,A -90.000,B 90.000,C 0.000} C_DIS
LIN {X 22.816,Y -35.308,Z -62.226,A -90.000,B 90.000,C 0.000} C_DIS
LIN {X 23.044,Y -35.308,Z -62.048,A -90.000,B 90.000,C 0.000} C_DIS
LIN {X 23.269,Y -35.308,Z -61.880,A -90.000,B 90.000,C 0.000} C_DIS
LIN {X 23.494,Y -35.308,Z -61.720,A -90.000,B 90.000,C 0.000} C_DIS
LIN {X 23.876,Y -35.308,Z -61.458,A -90.000,B 90.000,C 0.000} C_DIS
LIN {X 24.034,Y -35.308,Z -61.350,A -90.000,B 90.000,C 0.000} C_DIS
LIN {X 24.269,Y -35.308,Z -61.199,A -90.000,B 90.000,C 0.000} C_DIS
LIN {X 24.513,Y -35.308,Z -61.049,A -90.000,B 90.000,C 0.000} C_DIS
LIN {X 24.831,Y -35.308,Z -60.865,A -90.000,B 90.000,C 0.000} C_DIS
LIN {X 25.100,Y -35.308,Z -60.718,A -90.000,B 90.000,C 0.000} C_DIS
LIN {X 25.429,Y -35.308,Z -60.545,A -90.000,B 90.000,C 0.000} C_DIS
LIN {X 25.727,Y -35.308,Z -60.394,A -90.000,B 90.000,C 0.000} C_DIS
LIN {X 26.044,Y -35.308,Z -60.235,A -90.000,B 90.000,C 0.000} C_DIS
LIN {X 26.434,Y -35.308,Z -60.051,A -90.000,B 90.000,C 0.000} C_DIS
LIN {X 26.464,Y -35.308,Z -60.039,A -90.000,B 90.000,C 0.000} C_DIS
LIN {X 26.405,Y -35.308,Z -59.643,A -90.000,B 90.000,C 0.000} C_DIS
LIN {X 26.372,Y -35.308,Z -59.320,A -90.000,B 90.000,C 0.000} C_DIS
LIN {X 26.344,Y -35.308,Z -58.844,A -90.000,B 90.000,C 0.000} C_DIS
LIN {X 26.338,Y -35.308,Z -58.609,A -90.000,B 90.000,C 0.000} C_DIS
LIN {X 26.332,Y -35.308,Z -58.198,A -90.000,B 90.000,C 0.000} C_DIS
LIN {X 26.375,Y -35.308,Z -57.713,A -90.000,B 90.000,C 0.000} C_DIS
LIN {X 26.389,Y -35.308,Z -57.599,A -90.000,B 90.000,C 0.000} C_DIS
LIN {X 26.458,Y -35.308,Z -57.257,A -90.000,B 90.000,C 0.000} C_DIS
LIN {X 26.485,Y -35.308,Z -57.145,A -90.000,B 90.000,C 0.000} C_DIS
LIN {X 26.566,Y -35.308,Z -56.866,A -90.000,B 90.000,C 0.000} C_DIS
LIN {X 26.719,Y -35.308,Z -56.437,A -90.000,B 90.000,C 0.000} C_DIS
LIN {X 26.918,Y -35.308,Z -56.027,A -90.000,B 90.000,C 0.000} C_DIS
LIN {X 27.008,Y -35.308,Z -55.860,A -90.000,B 90.000,C 0.000} C_DIS
LIN {X 27.152,Y -35.308,Z -55.629,A -90.000,B 90.000,C 0.000} C_DIS
LIN {X 27.251,Y -35.308,Z -55.475,A -90.000,B 90.000,C 0.000} C_DIS
LIN {X 27.398,Y -35.308,Z -55.263,A -90.000,B 90.000,C 0.000} C_DIS
LIN {X 27.683,Y -35.308,Z -54.927,A -90.000,B 90.000,C 0.000} C_DIS
LIN {X 28.005,Y -35.308,Z -54.625,A -90.000,B 90.000,C 0.000} C_DIS
LIN {X 28.358,Y -35.308,Z -54.362,A -90.000,B 90.000,C 0.000} C_DIS
LIN {X 28.739,Y -35.308,Z -54.140,A -90.000,B 90.000,C 0.000} C_DIS
LIN {X 28.939,Y -35.308,Z -54.040,A -90.000,B 90.000,C 0.000} C_DIS
LIN {X 29.343,Y -35.308,Z -53.863,A -90.000,B 90.000,C 0.000} C_DIS
LIN {X 29.764,Y -35.308,Z -53.732,A -90.000,B 90.000,C 0.000} C_DIS
LIN {X 30.078,Y -35.308,Z -53.664,A -90.000,B 90.000,C 0.000} C_DIS
LIN {X 30.498,Y -35.308,Z -53.584,A -90.000,B 90.000,C 0.000} C_DIS
LIN {X 30.522,Y -35.308,Z -53.359,A -90.000,B 90.000,C 0.000} C_DIS
LIN {X 30.582,Y -35.308,Z -52.922,A -90.000,B 90.000,C 0.000} C_DIS
LIN {X 30.691,Y -35.308,Z -52.495,A -90.000,B 90.000,C 0.000} C_DIS
LIN {X 30.798,Y -35.308,Z -52.132,A -90.000,B 90.000,C 0.000} C_DIS
LIN {X 30.884,Y -35.308,Z -51.889,A -90.000,B 90.000,C 0.000} C_DIS
LIN {X 31.041,Y -35.308,Z -51.477,A -90.000,B 90.000,C 0.000} C_DIS
LIN {X 31.244,Y -35.308,Z -51.085,A -90.000,B 90.000,C 0.000} C_DIS
LIN {X 31.496,Y -35.308,Z -50.630,A -90.000,B 90.000,C 0.000} C_DIS
LIN {X 31.605,Y -35.308,Z -50.442,A -90.000,B 90.000,C 0.000} C_DIS
LIN {X 31.845,Y -35.308,Z -50.093,A -90.000,B 90.000,C 0.000} C_DIS
LIN {X 32.241,Y -35.308,Z -49.644,A -90.000,B 90.000,C 0.000} C_DIS
LIN {X 32.568,Y -35.308,Z -49.277,A -90.000,B 90.000,C 0.000} C_DIS
LIN {X 32.886,Y -35.308,Z -48.992,A -90.000,B 90.000,C 0.000} C_DIS
LIN {X 33.233,Y -35.308,Z -48.746,A -90.000,B 90.000,C 0.000} C_DIS
LIN {X 33.856,Y -35.308,Z -48.339,A -90.000,B 90.000,C 0.000} C_DIS
LIN {X 34.229,Y -35.308,Z -48.138,A -90.000,B 90.000,C 0.000} C_DIS
LIN {X 34.647,Y -35.308,Z -47.973,A -90.000,B 90.000,C 0.000} C_DIS
LIN {X 35.068,Y -35.308,Z -47.843,A -90.000,B 90.000,C 0.000} C_DIS
LIN {X 35.236,Y -35.308,Z -47.802,A -90.000,B 90.000,C 0.000} C_DIS
LIN {X 35.891,Y -35.308,Z -47.610,A -90.000,B 90.000,C 0.000} C_DIS
LIN {X 36.325,Y -35.308,Z -47.528,A -90.000,B 90.000,C 0.000} C_DIS
LIN {X 36.764,Y -35.308,Z -47.496,A -90.000,B 90.000,C 0.000} C_DIS
LIN {X 37.363,Y -35.308,Z -47.484,A -90.000,B 90.000,C 0.000} C_DIS
LIN {X 37.817,Y -35.308,Z -47.470,A -90.000,B 90.000,C 0.000} C_DIS
LIN {X 38.333,Y -35.308,Z -47.465,A -90.000,B 90.000,C 0.000} C_DIS
LIN {X 38.787,Y -35.308,Z -47.506,A -90.000,B 90.000,C 0.000} C_DIS
LIN {X 39.370,Y -35.308,Z -47.598,A -90.000,B 90.000,C 0.000} C_DIS
LIN {X 40.151,Y -35.308,Z -47.744,A -90.000,B 90.000,C 0.000} C_DIS
LIN {X 40.549,Y -35.308,Z -47.824,A -90.000,B 90.000,C 0.000} C_DIS
LIN {X 40.684,Y -35.308,Z -47.856,A -90.000,B 90.000,C 0.000} C_DIS
LIN {X 41.986,Y -35.308,Z -48.238,A -90.000,B 90.000,C 0.000} C_DIS
LIN {X 42.827,Y -35.308,Z -48.444,A -90.000,B 90.000,C 0.000} C_DIS
LIN {X 43.483,Y -35.308,Z -48.512,A -90.000,B 90.000,C 0.000} C_DIS
LIN {X 44.259,Y -35.308,Z -48.403,A -90.000,B 90.000,C 0.000} C_DIS
LIN {X 44.949,Y -35.308,Z -48.264,A -90.000,B 90.000,C 0.000} C_DIS
LIN {X 45.823,Y -35.308,Z -48.069,A -90.000,B 90.000,C 0.000} C_DIS
LIN {X 46.280,Y -35.308,Z -48.005,A -90.000,B 90.000,C 0.000} C_DIS
LIN {X 47.255,Y -35.308,Z -47.896,A -90.000,B 90.000,C 0.000} C_DIS
LIN {X 48.074,Y -35.308,Z -47.777,A -90.000,B 90.000,C 0.000} C_DIS
LIN {X 48.497,Y -35.308,Z -47.767,A -90.000,B 90.000,C 0.000} C_DIS
LIN {X 48.993,Y -35.308,Z -47.815,A -90.000,B 90.000,C 0.000} C_DIS
LIN {X 51.093,Y -35.308,Z -48.054,A -90.000,B 90.000,C 0.000} C_DIS
LIN {X 51.504,Y -35.308,Z -48.093,A -90.000,B 90.000,C 0.000} C_DIS
LIN {X 51.766,Y -35.308,Z -48.139,A -90.000,B 90.000,C 0.000} C_DIS
LIN {X 52.006,Y -35.308,Z -48.191,A -90.000,B 90.000,C 0.000} C_DIS
LIN {X 52.185,Y -35.308,Z -48.239,A -90.000,B 90.000,C 0.000} C_DIS
LIN {X 52.417,Y -35.308,Z -48.319,A -90.000,B 90.000,C 0.000} C_DIS
LIN {X 52.589,Y -35.308,Z -48.388,A -90.000,B 90.000,C 0.000} C_DIS
LIN {X 52.810,Y -35.308,Z -48.495,A -90.000,B 90.000,C 0.000} C_DIS
LIN {X 52.973,Y -35.308,Z -48.582,A -90.000,B 90.000,C 0.000} C_DIS
LIN {X 54.792,Y -35.308,Z -49.747,A -90.000,B 90.000,C 0.000} C_DIS
LIN {X 56.047,Y -35.308,Z -50.582,A -90.000,B 90.000,C 0.000} C_DIS
LIN {X 56.272,Y -35.308,Z -50.738,A -90.000,B 90.000,C 0.000} C_DIS
LIN {X 56.411,Y -35.308,Z -50.840,A -90.000,B 90.000,C 0.000} C_DIS
LIN {X 58.818,Y -35.308,Z -52.892,A -90.000,B 90.000,C 0.000} C_DIS
LIN {X 59.039,Y -35.308,Z -53.085,A -90.000,B 90.000,C 0.000} C_DIS
LIN {X 59.151,Y -35.308,Z -53.189,A -90.000,B 90.000,C 0.000} C_DIS
LIN {X 60.234,Y -35.308,Z -54.223,A -90.000,B 90.000,C 0.000} C_DIS
LIN {X 61.288,Y -35.308,Z -55.260,A -90.000,B 90.000,C 0.000} C_DIS
LIN {X 62.570,Y -35.308,Z -56.601,A -90.000,B 90.000,C 0.000} C_DIS
LIN {X 63.609,Y -35.308,Z -57.726,A -90.000,B 90.000,C 0.000} C_DIS
LIN {X 64.523,Y -35.308,Z -58.738,A -90.000,B 90.000,C 0.000} C_DIS
LIN {X 65.687,Y -35.308,Z -60.006,A -90.000,B 90.000,C 0.000} C_DIS
LIN {X 66.403,Y -35.308,Z -60.817,A -90.000,B 90.000,C 0.000} C_DIS
LIN {X 67.045,Y -35.308,Z -61.564,A -90.000,B 90.000,C 0.000} C_DIS
LIN {X 67.299,Y -35.308,Z -61.877,A -90.000,B 90.000,C 0.000} C_DIS
LIN {X 69.467,Y -35.308,Z -64.801,A -90.000,B 90.000,C 0.000} C_DIS
LIN {X 70.998,Y -35.308,Z -66.881,A -90.000,B 90.000,C 0.000} C_DIS
LIN {X 71.095,Y -35.308,Z -67.017,A -90.000,B 90.000,C 0.000} C_DIS
LIN {X 71.269,Y -35.308,Z -67.217,A -90.000,B 90.000,C 0.000} C_DIS
LIN {X 71.956,Y -35.308,Z -68.047,A -90.000,B 90.000,C 0.000} C_DIS
LIN {X 72.108,Y -35.308,Z -68.204,A -90.000,B 90.000,C 0.000} C_DIS
LIN {X 72.618,Y -35.308,Z -68.818,A -90.000,B 90.000,C 0.000} C_DIS
LIN {X 73.347,Y -35.308,Z -69.527,A -90.000,B 90.000,C 0.000} C_DIS
LIN {X 73.435,Y -35.308,Z -69.631,A -90.000,B 90.000,C 0.000} C_DIS
LIN {X 73.533,Y -35.308,Z -69.726,A -90.000,B 90.000,C 0.000} C_DIS
LIN {X 73.702,Y -35.308,Z -69.890,A -90.000,B 90.000,C 0.000} C_DIS
LIN {X 74.491,Y -35.308,Z -70.670,A -90.000,B 90.000,C 0.000} C_DIS
LIN {X 75.226,Y -35.308,Z -71.403,A -90.000,B 90.000,C 0.000} C_DIS
LIN {X 75.554,Y -35.308,Z -71.736,A -90.000,B 90.000,C 0.000} C_DIS
LIN {X 75.682,Y -35.308,Z -71.869,A -90.000,B 90.000,C 0.000} C_DIS
LIN {X 76.444,Y -35.308,Z -72.712,A -90.000,B 90.000,C 0.000} C_DIS
LIN {X 76.882,Y -35.308,Z -73.205,A -90.000,B 90.000,C 0.000} C_DIS
LIN {X 77.181,Y -35.308,Z -73.548,A -90.000,B 90.000,C 0.000} C_DIS
LIN {X 77.659,Y -35.308,Z -74.104,A -90.000,B 90.000,C 0.000} C_DIS
LIN {X 77.743,Y -35.308,Z -73.625,A -90.000,B 90.000,C 0.000} C_DIS
LIN {X 77.847,Y -35.308,Z -73.149,A -90.000,B 90.000,C 0.000} C_DIS
LIN {X 77.996,Y -35.308,Z -72.490,A -90.000,B 90.000,C 0.000} C_DIS
LIN {X 78.121,Y -35.308,Z -71.990,A -90.000,B 90.000,C 0.000} C_DIS
LIN {X 78.173,Y -35.308,Z -71.793,A -90.000,B 90.000,C 0.000} C_DIS
LIN {X 78.642,Y -35.308,Z -70.361,A -90.000,B 90.000,C 0.000} C_DIS
LIN {X 78.804,Y -35.308,Z -69.881,A -90.000,B 90.000,C 0.000} C_DIS
LIN {X 79.205,Y -35.308,Z -68.728,A -90.000,B 90.000,C 0.000} C_DIS
LIN {X 79.796,Y -35.308,Z -67.247,A -90.000,B 90.000,C 0.000} C_DIS
LIN {X 80.445,Y -35.308,Z -65.774,A -90.000,B 90.000,C 0.000} C_DIS
LIN {X 80.645,Y -35.308,Z -65.334,A -90.000,B 90.000,C 0.000} C_DIS
LIN {X 81.438,Y -35.308,Z -63.804,A -90.000,B 90.000,C 0.000} C_DIS
LIN {X 81.684,Y -35.308,Z -63.383,A -90.000,B 90.000,C 0.000} C_DIS
LIN {X 82.705,Y -35.308,Z -61.742,A -90.000,B 90.000,C 0.000} C_DIS
LIN {X 84.243,Y -35.308,Z -59.630,A -90.000,B 90.000,C 0.000} C_DIS
LIN {X 84.612,Y -35.308,Z -59.191,A -90.000,B 90.000,C 0.000} C_DIS
LIN {X 85.732,Y -35.308,Z -57.856,A -90.000,B 90.000,C 0.000} C_DIS
LIN {X 86.059,Y -35.308,Z -57.494,A -90.000,B 90.000,C 0.000} C_DIS
LIN {X 87.795,Y -35.308,Z -55.685,A -90.000,B 90.000,C 0.000} C_DIS
LIN {X 89.946,Y -35.308,Z -53.718,A -90.000,B 90.000,C 0.000} C_DIS
LIN {X 90.164,Y -35.308,Z -53.522,A -90.000,B 90.000,C 0.000} C_DIS
LIN {X 92.263,Y -35.308,Z -51.722,A -90.000,B 90.000,C 0.000} C_DIS
LIN {X 94.367,Y -35.308,Z -49.945,A -90.000,B 90.000,C 0.000} C_DIS
LIN {X 96.081,Y -35.308,Z -48.442,A -90.000,B 90.000,C 0.000} C_DIS
LIN {X 97.648,Y -35.308,Z -46.921,A -90.000,B 90.000,C 0.000} C_DIS
LIN {X 98.544,Y -35.308,Z -45.976,A -90.000,B 90.000,C 0.000} C_DIS
LIN {X 98.363,Y -35.308,Z -45.464,A -90.000,B 90.000,C 0.000} C_DIS
LIN {X 98.292,Y -35.308,Z -45.153,A -90.000,B 90.000,C 0.000} C_DIS
LIN {X 98.273,Y -35.308,Z -44.949,A -90.000,B 90.000,C 0.000} C_DIS
LIN {X 98.269,Y -35.308,Z -44.867,A -90.000,B 90.000,C 0.000} C_DIS
LIN {X 98.241,Y -35.308,Z -44.669,A -90.000,B 90.000,C 0.000} C_DIS
LIN {X 98.220,Y -35.308,Z -44.351,A -90.000,B 90.000,C 0.000} C_DIS
LIN {X 98.222,Y -35.308,Z -44.117,A -90.000,B 90.000,C 0.000} C_DIS
LIN {X 98.251,Y -35.308,Z -43.767,A -90.000,B 90.000,C 0.000} C_DIS
LIN {X 98.330,Y -35.308,Z -43.424,A -90.000,B 90.000,C 0.000} C_DIS
LIN {X 98.528,Y -35.308,Z -42.828,A -90.000,B 90.000,C 0.000} C_DIS
LIN {X 98.694,Y -35.308,Z -42.476,A -90.000,B 90.000,C 0.000} C_DIS
LIN {X 98.971,Y -35.308,Z -41.945,A -90.000,B 90.000,C 0.000} C_DIS
LIN {X 99.418,Y -35.308,Z -41.289,A -90.000,B 90.000,C 0.000} C_DIS
LIN {X 99.499,Y -35.308,Z -41.179,A -90.000,B 90.000,C 0.000} C_DIS
LIN {X 99.560,Y -35.308,Z -41.092,A -90.000,B 90.000,C 0.000} C_DIS
LIN {X 99.698,Y -35.308,Z -40.902,A -90.000,B 90.000,C 0.000} C_DIS
LIN {X 99.805,Y -35.308,Z -40.771,A -90.000,B 90.000,C 0.000} C_DIS
LIN {X 100.084,Y -35.308,Z -40.453,A -90.000,B 90.000,C 0.000} C_DIS
LIN {X 100.547,Y -35.308,Z -39.966,A -90.000,B 90.000,C 0.000} C_DIS
LIN {X 100.868,Y -35.308,Z -39.664,A -90.000,B 90.000,C 0.000} C_DIS
LIN {X 100.987,Y -35.308,Z -39.557,A -90.000,B 90.000,C 0.000} C_DIS
LIN {X 101.188,Y -35.308,Z -39.361,A -90.000,B 90.000,C 0.000} C_DIS
LIN {X 101.359,Y -35.308,Z -39.216,A -90.000,B 90.000,C 0.000} C_DIS
LIN {X 102.150,Y -35.308,Z -38.580,A -90.000,B 90.000,C 0.000} C_DIS
LIN {X 102.529,Y -35.308,Z -38.307,A -90.000,B 90.000,C 0.000} C_DIS
LIN {X 102.904,Y -35.308,Z -38.046,A -90.000,B 90.000,C 0.000} C_DIS
LIN {X 103.439,Y -35.308,Z -37.696,A -90.000,B 90.000,C 0.000} C_DIS
LIN {X 104.294,Y -35.308,Z -37.184,A -90.000,B 90.000,C 0.000} C_DIS
LIN {X 104.456,Y -35.308,Z -37.097,A -90.000,B 90.000,C 0.000} C_DIS
LIN {X 105.066,Y -35.308,Z -36.797,A -90.000,B 90.000,C 0.000} C_DIS
LIN {X 105.305,Y -35.308,Z -36.682,A -90.000,B 90.000,C 0.000} C_DIS
LIN {X 105.504,Y -35.308,Z -36.590,A -90.000,B 90.000,C 0.000} C_DIS
LIN {X 106.262,Y -35.308,Z -36.255,A -90.000,B 90.000,C 0.000} C_DIS
LIN {X 106.502,Y -35.308,Z -36.160,A -90.000,B 90.000,C 0.000} C_DIS
LIN {X 106.852,Y -35.308,Z -36.003,A -90.000,B 90.000,C 0.000} C_DIS
LIN {X 107.404,Y -35.308,Z -35.786,A -90.000,B 90.000,C 0.000} C_DIS
LIN {X 107.845,Y -35.308,Z -35.629,A -90.000,B 90.000,C 0.000} C_DIS
LIN {X 108.305,Y -35.308,Z -35.472,A -90.000,B 90.000,C 0.000} C_DIS
LIN {X 108.737,Y -35.308,Z -35.349,A -90.000,B 90.000,C 0.000} C_DIS
LIN {X 109.212,Y -35.308,Z -35.240,A -90.000,B 90.000,C 0.000} C_DIS
LIN {X 109.619,Y -35.308,Z -35.179,A -90.000,B 90.000,C 0.000} C_DIS
LIN {X 110.103,Y -35.308,Z -35.120,A -90.000,B 90.000,C 0.000} C_DIS
LIN {X 110.591,Y -35.308,Z -35.111,A -90.000,B 90.000,C 0.000} C_DIS
LIN {X 110.949,Y -35.308,Z -35.117,A -90.000,B 90.000,C 0.000} C_DIS
LIN {X 111.435,Y -35.308,Z -35.158,A -90.000,B 90.000,C 0.000} C_DIS
LIN {X 112.069,Y -35.308,Z -35.277,A -90.000,B 90.000,C 0.000} C_DIS
LIN {X 112.408,Y -35.308,Z -35.363,A -90.000,B 90.000,C 0.000} C_DIS
LIN {X 112.874,Y -35.308,Z -35.502,A -90.000,B 90.000,C 0.000} C_DIS
LIN {X 113.059,Y -35.308,Z -35.562,A -90.000,B 90.000,C 0.000} C_DIS
LIN {X 113.511,Y -35.308,Z -35.749,A -90.000,B 90.000,C 0.000} C_DIS
LIN {X 113.987,Y -35.308,Z -35.977,A -90.000,B 90.000,C 0.000} C_DIS
LIN {X 114.411,Y -35.308,Z -36.206,A -90.000,B 90.000,C 0.000} C_DIS
LIN {X 114.550,Y -35.308,Z -36.292,A -90.000,B 90.000,C 0.000} C_DIS
LIN {X 114.946,Y -35.308,Z -36.562,A -90.000,B 90.000,C 0.000} C_DIS
LIN {X 115.058,Y -35.308,Z -36.651,A -90.000,B 90.000,C 0.000} C_DIS
LIN {X 115.423,Y -35.308,Z -36.958,A -90.000,B 90.000,C 0.000} C_DIS
LIN {X 115.524,Y -35.308,Z -37.050,A -90.000,B 90.000,C 0.000} C_DIS
LIN {X 115.859,Y -35.308,Z -37.397,A -90.000,B 90.000,C 0.000} C_DIS
LIN {X 116.077,Y -35.308,Z -37.628,A -90.000,B 90.000,C 0.000} C_DIS
LIN {X 116.439,Y -35.308,Z -38.088,A -90.000,B 90.000,C 0.000} C_DIS
LIN {X 116.700,Y -35.308,Z -38.500,A -90.000,B 90.000,C 0.000} C_DIS
LIN {X 116.922,Y -35.308,Z -38.948,A -90.000,B 90.000,C 0.000} C_DIS
LIN {X 117.057,Y -35.308,Z -39.246,A -90.000,B 90.000,C 0.000} C_DIS
LIN {X 117.096,Y -35.308,Z -39.342,A -90.000,B 90.000,C 0.000} C_DIS
LIN {X 117.260,Y -35.308,Z -39.781,A -90.000,B 90.000,C 0.000} C_DIS
LIN {X 117.387,Y -35.308,Z -40.266,A -90.000,B 90.000,C 0.000} C_DIS
LIN {X 117.464,Y -35.308,Z -40.606,A -90.000,B 90.000,C 0.000} C_DIS
LIN {X 117.538,Y -35.308,Z -41.090,A -90.000,B 90.000,C 0.000} C_DIS
LIN {X 117.594,Y -35.308,Z -41.507,A -90.000,B 90.000,C 0.000} C_DIS
LIN {X 117.631,Y -35.308,Z -41.891,A -90.000,B 90.000,C 0.000} C_DIS
LIN {X 117.656,Y -35.308,Z -42.373,A -90.000,B 90.000,C 0.000} C_DIS
LIN {X 117.668,Y -35.308,Z -42.690,A -90.000,B 90.000,C 0.000} C_DIS
LIN {X 117.665,Y -35.308,Z -42.850,A -90.000,B 90.000,C 0.000} C_DIS
LIN {X 117.651,Y -35.308,Z -43.213,A -90.000,B 90.000,C 0.000} C_DIS
LIN {X 117.609,Y -35.308,Z -43.701,A -90.000,B 90.000,C 0.000} C_DIS
LIN {X 117.565,Y -35.308,Z -44.130,A -90.000,B 90.000,C 0.000} C_DIS
LIN {X 117.487,Y -35.308,Z -44.645,A -90.000,B 90.000,C 0.000} C_DIS
LIN {X 117.396,Y -35.308,Z -45.128,A -90.000,B 90.000,C 0.000} C_DIS
LIN {X 117.258,Y -35.308,Z -45.747,A -90.000,B 90.000,C 0.000} C_DIS
LIN {X 117.120,Y -35.308,Z -46.210,A -90.000,B 90.000,C 0.000} C_DIS
LIN {X 116.899,Y -35.308,Z -46.941,A -90.000,B 90.000,C 0.000} C_DIS
LIN {X 116.556,Y -35.308,Z -47.832,A -90.000,B 90.000,C 0.000} C_DIS
LIN {X 116.370,Y -35.308,Z -48.283,A -90.000,B 90.000,C 0.000} C_DIS
LIN {X 115.872,Y -35.308,Z -49.353,A -90.000,B 90.000,C 0.000} C_DIS
LIN {X 115.513,Y -35.308,Z -50.071,A -90.000,B 90.000,C 0.000} C_DIS
LIN {X 114.841,Y -35.308,Z -51.387,A -90.000,B 90.000,C 0.000} C_DIS
LIN {X 114.626,Y -35.308,Z -51.805,A -90.000,B 90.000,C 0.000} C_DIS
LIN {X 113.947,Y -35.308,Z -53.175,A -90.000,B 90.000,C 0.000} C_DIS
LIN {X 113.284,Y -35.308,Z -54.614,A -90.000,B 90.000,C 0.000} C_DIS
LIN {X 112.688,Y -35.308,Z -56.016,A -90.000,B 90.000,C 0.000} C_DIS
LIN {X 112.185,Y -35.308,Z -57.324,A -90.000,B 90.000,C 0.000} C_DIS
LIN {X 111.587,Y -35.308,Z -59.065,A -90.000,B 90.000,C 0.000} C_DIS
LIN {X 111.015,Y -35.308,Z -60.937,A -90.000,B 90.000,C 0.000} C_DIS
LIN {X 110.413,Y -35.308,Z -62.968,A -90.000,B 90.000,C 0.000} C_DIS
LIN {X 109.804,Y -35.308,Z -64.894,A -90.000,B 90.000,C 0.000} C_DIS
LIN {X 109.352,Y -35.308,Z -66.208,A -90.000,B 90.000,C 0.000} C_DIS
LIN {X 108.885,Y -35.308,Z -67.529,A -90.000,B 90.000,C 0.000} C_DIS
LIN {X 108.648,Y -35.308,Z -68.139,A -90.000,B 90.000,C 0.000} C_DIS
LIN {X 107.938,Y -35.308,Z -69.948,A -90.000,B 90.000,C 0.000} C_DIS
LIN {X 107.195,Y -35.308,Z -71.714,A -90.000,B 90.000,C 0.000} C_DIS
LIN {X 106.905,Y -35.308,Z -72.395,A -90.000,B 90.000,C 0.000} C_DIS
LIN {X 106.174,Y -35.308,Z -74.000,A -90.000,B 90.000,C 0.000} C_DIS
LIN {X 106.051,Y -35.308,Z -74.265,A -90.000,B 90.000,C 0.000} C_DIS
LIN {X 105.618,Y -35.308,Z -75.189,A -90.000,B 90.000,C 0.000} C_DIS
LIN {X 104.514,Y -35.308,Z -77.348,A -90.000,B 90.000,C 0.000} C_DIS
LIN {X 103.437,Y -35.308,Z -79.232,A -90.000,B 90.000,C 0.000} C_DIS
LIN {X 103.190,Y -35.308,Z -79.647,A -90.000,B 90.000,C 0.000} C_DIS
LIN {X 102.158,Y -35.308,Z -81.287,A -90.000,B 90.000,C 0.000} C_DIS
LIN {X 101.930,Y -35.308,Z -81.622,A -90.000,B 90.000,C 0.000} C_DIS
LIN {X 101.183,Y -35.308,Z -82.703,A -90.000,B 90.000,C 0.000} C_DIS
LIN {X 100.610,Y -35.308,Z -83.494,A -90.000,B 90.000,C 0.000} C_DIS
LIN {X 99.352,Y -35.308,Z -85.238,A -90.000,B 90.000,C 0.000} C_DIS
LIN {X 98.753,Y -35.308,Z -86.065,A -90.000,B 90.000,C 0.000} C_DIS
LIN {X 97.638,Y -35.308,Z -87.568,A -90.000,B 90.000,C 0.000} C_DIS
LIN {X 97.174,Y -35.308,Z -88.169,A -90.000,B 90.000,C 0.000} C_DIS
LIN {X 97.069,Y -35.308,Z -88.406,A -90.000,B 90.000,C 0.000} C_DIS
LIN {X 96.966,Y -35.308,Z -88.809,A -90.000,B 90.000,C 0.000} C_DIS
LIN {X 96.901,Y -35.308,Z -89.038,A -90.000,B 90.000,C 0.000} C_DIS
LIN {X 96.689,Y -35.308,Z -90.269,A -90.000,B 90.000,C 0.000} C_DIS
LIN {X 96.555,Y -35.308,Z -91.265,A -90.000,B 90.000,C 0.000} C_DIS
LIN {X 96.437,Y -35.308,Z -92.185,A -90.000,B 90.000,C 0.000} C_DIS
LIN {X 96.390,Y -35.308,Z -92.566,A -90.000,B 90.000,C 0.000} C_DIS
LIN {X 96.277,Y -35.308,Z -93.539,A -90.000,B 90.000,C 0.000} C_DIS
LIN {X 96.220,Y -35.308,Z -93.915,A -90.000,B 90.000,C 0.000} C_DIS
LIN {X 96.200,Y -35.308,Z -94.067,A -90.000,B 90.000,C 0.000} C_DIS
LIN {X 96.028,Y -35.308,Z -95.095,A -90.000,B 90.000,C 0.000} C_DIS
LIN {X 95.940,Y -35.308,Z -95.671,A -90.000,B 90.000,C 0.000} C_DIS
LIN {X 95.845,Y -35.308,Z -96.101,A -90.000,B 90.000,C 0.000} C_DIS
LIN {X 95.730,Y -35.308,Z -96.577,A -90.000,B 90.000,C 0.000} C_DIS
LIN {X 95.576,Y -35.308,Z -97.251,A -90.000,B 90.000,C 0.000} C_DIS
LIN {X 95.506,Y -35.308,Z -97.457,A -90.000,B 90.000,C 0.000} C_DIS
LIN {X 95.274,Y -35.308,Z -98.185,A -90.000,B 90.000,C 0.000} C_DIS
LIN {X 95.130,Y -35.308,Z -98.602,A -90.000,B 90.000,C 0.000} C_DIS
LIN {X 94.848,Y -35.308,Z -99.228,A -90.000,B 90.000,C 0.000} C_DIS
LIN {X 94.342,Y -35.308,Z -100.377,A -90.000,B 90.000,C 0.000} C_DIS
LIN {X 93.889,Y -35.308,Z -101.555,A -90.000,B 90.000,C 0.000} C_DIS
LIN {X 93.551,Y -35.308,Z -102.567,A -90.000,B 90.000,C 0.000} C_DIS
LIN {X 93.494,Y -35.308,Z -102.714,A -90.000,B 90.000,C 0.000} C_DIS
LIN {X 93.191,Y -35.308,Z -103.670,A -90.000,B 90.000,C 0.000} C_DIS
LIN {X 93.029,Y -35.308,Z -104.473,A -90.000,B 90.000,C 0.000} C_DIS
LIN {X 93.036,Y -35.308,Z -104.940,A -90.000,B 90.000,C 0.000} C_DIS
LIN {X 93.041,Y -35.308,Z -104.986,A -90.000,B 90.000,C 0.000} C_DIS
LIN {X 93.180,Y -35.308,Z -105.893,A -90.000,B 90.000,C 0.000} C_DIS
LIN {X 93.350,Y -35.308,Z -106.823,A -90.000,B 90.000,C 0.000} C_DIS
LIN {X 93.364,Y -35.308,Z -106.905,A -90.000,B 90.000,C 0.000} C_DIS
LIN {X 93.535,Y -35.308,Z -108.246,A -90.000,B 90.000,C 0.000} C_DIS
LIN {X 93.560,Y -35.308,Z -108.668,A -90.000,B 90.000,C 0.000} C_DIS
LIN {X 93.610,Y -35.308,Z -110.357,A -90.000,B 90.000,C 0.000} C_DIS
LIN {X 93.579,Y -35.308,Z -112.469,A -90.000,B 90.000,C 0.000} C_DIS
LIN {X 93.508,Y -35.308,Z -114.473,A -90.000,B 90.000,C 0.000} C_DIS
LIN {X 93.455,Y -35.308,Z -116.602,A -90.000,B 90.000,C 0.000} C_DIS
LIN {X 93.460,Y -35.308,Z -117.182,A -90.000,B 90.000,C 0.000} C_DIS
LIN {X 93.455,Y -35.308,Z -118.767,A -90.000,B 90.000,C 0.000} C_DIS
LIN {X 93.482,Y -35.308,Z -120.687,A -90.000,B 90.000,C 0.000} C_DIS
LIN {X 93.488,Y -35.308,Z -120.902,A -90.000,B 90.000,C 0.000} C_DIS
LIN {X 93.509,Y -35.308,Z -122.696,A -90.000,B 90.000,C 0.000} C_DIS
LIN {X 93.519,Y -35.308,Z -122.995,A -90.000,B 90.000,C 0.000} C_DIS
LIN {X 93.501,Y -35.308,Z -124.662,A -90.000,B 90.000,C 0.000} C_DIS
LIN {X 93.504,Y -35.308,Z -125.046,A -90.000,B 90.000,C 0.000} C_DIS
LIN {X 93.476,Y -35.308,Z -125.713,A -90.000,B 90.000,C 0.000} C_DIS
LIN {X 93.390,Y -35.308,Z -127.314,A -90.000,B 90.000,C 0.000} C_DIS
LIN {X 93.345,Y -35.308,Z -127.873,A -90.000,B 90.000,C 0.000} C_DIS
LIN {X 93.216,Y -35.308,Z -129.408,A -90.000,B 90.000,C 0.000} C_DIS
LIN {X 92.893,Y -35.308,Z -132.746,A -90.000,B 90.000,C 0.000} C_DIS
LIN {X 92.735,Y -35.308,Z -134.380,A -90.000,B 90.000,C 0.000} C_DIS
LIN {X 92.468,Y -35.308,Z -137.527,A -90.000,B 90.000,C 0.000} C_DIS
LIN {X 92.296,Y -35.308,Z -139.509,A -90.000,B 90.000,C 0.000} C_DIS
LIN {X 92.166,Y -35.308,Z -141.024,A -90.000,B 90.000,C 0.000} C_DIS
LIN {X 91.956,Y -35.308,Z -143.155,A -90.000,B 90.000,C 0.000} C_DIS
LIN {X 91.805,Y -35.308,Z -144.731,A -90.000,B 90.000,C 0.000} C_DIS
LIN {X 91.539,Y -35.308,Z -146.962,A -90.000,B 90.000,C 0.000} C_DIS
LIN {X 91.359,Y -35.308,Z -148.512,A -90.000,B 90.000,C 0.000} C_DIS
LIN {X 91.091,Y -35.308,Z -150.352,A -90.000,B 90.000,C 0.000} C_DIS
LIN {X 90.748,Y -35.308,Z -152.623,A -90.000,B 90.000,C 0.000} C_DIS
LIN {X 90.505,Y -35.308,Z -153.992,A -90.000,B 90.000,C 0.000} C_DIS
LIN {X 90.085,Y -35.308,Z -156.282,A -90.000,B 90.000,C 0.000} C_DIS
LIN {X 89.807,Y -35.308,Z -157.608,A -90.000,B 90.000,C 0.000} C_DIS
LIN {X 89.311,Y -35.308,Z -159.903,A -90.000,B 90.000,C 0.000} C_DIS
LIN {X 88.989,Y -35.308,Z -161.229,A -90.000,B 90.000,C 0.000} C_DIS
LIN {X 88.427,Y -35.308,Z -163.501,A -90.000,B 90.000,C 0.000} C_DIS
LIN {X 87.938,Y -35.308,Z -165.273,A -90.000,B 90.000,C 0.000} C_DIS
LIN {X 87.325,Y -35.308,Z -167.479,A -90.000,B 90.000,C 0.000} C_DIS
LIN {X 86.270,Y -35.308,Z -170.996,A -90.000,B 90.000,C 0.000} C_DIS
LIN {X 85.208,Y -35.308,Z -174.380,A -90.000,B 90.000,C 0.000} C_DIS
LIN {X 84.726,Y -35.308,Z -175.901,A -90.000,B 90.000,C 0.000} C_DIS
LIN {X 84.117,Y -35.308,Z -177.803,A -90.000,B 90.000,C 0.000} C_DIS
LIN {X 83.749,Y -35.308,Z -178.964,A -90.000,B 90.000,C 0.000} C_DIS
LIN {X 83.303,Y -35.308,Z -180.407,A -90.000,B 90.000,C 0.000} C_DIS
LIN {X 83.003,Y -35.308,Z -181.357,A -90.000,B 90.000,C 0.000} C_DIS
LIN {X 82.461,Y -35.308,Z -183.149,A -90.000,B 90.000,C 0.000} C_DIS
LIN {X 82.143,Y -35.308,Z -184.155,A -90.000,B 90.000,C 0.000} C_DIS
LIN {X 81.657,Y -35.308,Z -185.768,A -90.000,B 90.000,C 0.000} C_DIS
LIN {X 81.316,Y -35.308,Z -186.841,A -90.000,B 90.000,C 0.000} C_DIS
LIN {X 80.878,Y -35.308,Z -188.284,A -90.000,B 90.000,C 0.000} C_DIS
LIN {X 80.506,Y -35.308,Z -189.438,A -90.000,B 90.000,C 0.000} C_DIS
LIN {X 80.102,Y -35.308,Z -190.743,A -90.000,B 90.000,C 0.000} C_DIS
LIN {X 79.668,Y -35.308,Z -192.046,A -90.000,B 90.000,C 0.000} C_DIS
LIN {X 79.256,Y -35.308,Z -193.316,A -90.000,B 90.000,C 0.000} C_DIS
LIN {X 79.122,Y -35.308,Z -193.718,A -90.000,B 90.000,C 0.000} C_DIS
LIN {X 78.587,Y -35.308,Z -195.256,A -90.000,B 90.000,C 0.000} C_DIS
LIN {X 78.133,Y -35.308,Z -196.576,A -90.000,B 90.000,C 0.000} C_DIS
LIN {X 76.928,Y -35.308,Z -199.889,A -90.000,B 90.000,C 0.000} C_DIS
LIN {X 76.055,Y -35.308,Z -202.193,A -90.000,B 90.000,C 0.000} C_DIS
LIN {X 75.432,Y -35.308,Z -203.828,A -90.000,B 90.000,C 0.000} C_DIS
LIN {X 74.382,Y -35.308,Z -206.498,A -90.000,B 90.000,C 0.000} C_DIS
LIN {X 73.680,Y -35.308,Z -208.267,A -90.000,B 90.000,C 0.000} C_DIS
LIN {X 72.467,Y -35.308,Z -211.238,A -90.000,B 90.000,C 0.000} C_DIS
LIN {X 71.669,Y -35.308,Z -213.167,A -90.000,B 90.000,C 0.000} C_DIS
LIN {X 70.342,Y -35.308,Z -216.289,A -90.000,B 90.000,C 0.000} C_DIS
LIN {X 69.541,Y -35.308,Z -218.151,A -90.000,B 90.000,C 0.000} C_DIS
LIN {X 68.718,Y -35.308,Z -219.979,A -90.000,B 90.000,C 0.000} C_DIS
LIN {X 67.210,Y -35.308,Z -223.372,A -90.000,B 90.000,C 0.000} C_DIS
LIN {X 66.378,Y -35.308,Z -225.138,A -90.000,B 90.000,C 0.000} C_DIS
LIN {X 64.700,Y -35.308,Z -228.779,A -90.000,B 90.000,C 0.000} C_DIS
LIN {X 64.577,Y -35.308,Z -229.041,A -90.000,B 90.000,C 0.000} C_DIS
LIN {X 63.793,Y -35.308,Z -230.628,A -90.000,B 90.000,C 0.000} C_DIS
LIN {X 61.978,Y -35.308,Z -234.454,A -90.000,B 90.000,C 0.000} C_DIS
LIN {X 61.616,Y -35.308,Z -235.154,A -90.000,B 90.000,C 0.000} C_DIS
LIN {X 59.394,Y -35.308,Z -239.742,A -90.000,B 90.000,C 0.000} C_DIS
LIN {X 58.786,Y -35.308,Z -240.975,A -90.000,B 90.000,C 0.000} C_DIS
LIN {X 57.531,Y -35.308,Z -243.561,A -90.000,B 90.000,C 0.000} C_DIS
LIN {X 57.531,Y -60.000,Z -243.561,A -90.000,B 90.000,C 0.000} C_DIS
LIN {X 114.587,Y -60.000,Z -51.910,A -90.000,B 90.000,C 0.000} C_DIS
LIN {X 114.587,Y -33.308,Z -51.910,A -90.000,B 90.000,C 0.000} C_DIS
LIN {X 113.934,Y -33.308,Z -53.246,A -90.000,B 90.000,C 0.000} C_DIS
LIN {X 113.269,Y -33.309,Z -54.704,A -90.000,B 90.000,C 0.000} C_DIS
LIN {X 112.799,Y -33.309,Z -55.830,A -90.000,B 90.000,C 0.000} C_DIS
LIN {X 112.206,Y -33.309,Z -57.409,A -90.000,B 90.000,C 0.000} C_DIS
LIN {X 111.674,Y -33.309,Z -59.009,A -90.000,B 90.000,C 0.000} C_DIS
LIN {X 111.248,Y -33.310,Z -60.487,A -90.000,B 90.000,C 0.000} C_DIS
LIN {X 110.729,Y -33.313,Z -62.394,A -90.000,B 90.000,C 0.000} C_DIS
LIN {X 110.160,Y -33.318,Z -64.411,A -90.000,B 90.000,C 0.000} C_DIS
LIN {X 110.020,Y -33.319,Z -64.884,A -90.000,B 90.000,C 0.000} C_DIS
LIN {X 109.346,Y -33.324,Z -66.979,A -90.000,B 90.000,C 0.000} C_DIS
LIN {X 108.993,Y -33.323,Z -67.921,A -90.000,B 90.000,C 0.000} C_DIS
LIN {X 108.437,Y -33.326,Z -69.396,A -90.000,B 90.000,C 0.000} C_DIS
LIN {X 108.263,Y -33.326,Z -69.839,A -90.000,B 90.000,C 0.000} C_DIS
LIN {X 107.769,Y -33.327,Z -71.054,A -90.000,B 90.000,C 0.000} C_DIS
LIN {X 107.253,Y -33.329,Z -72.308,A -90.000,B 90.000,C 0.000} C_DIS
LIN {X 106.188,Y -33.334,Z -74.724,A -90.000,B 90.000,C 0.000} C_DIS
LIN {X 105.887,Y -33.331,Z -75.327,A -90.000,B 90.000,C 0.000} C_DIS
LIN {X 105.107,Y -33.334,Z -76.885,A -90.000,B 90.000,C 0.000} C_DIS
LIN {X 105.056,Y -33.334,Z -76.985,A -90.000,B 90.000,C 0.000} C_DIS
LIN {X 104.874,Y -33.333,Z -77.335,A -90.000,B 90.000,C 0.000} C_DIS
LIN {X 103.829,Y -33.336,Z -79.213,A -90.000,B 90.000,C 0.000} C_DIS
LIN {X 103.460,Y -33.334,Z -79.817,A -90.000,B 90.000,C 0.000} C_DIS
LIN {X 102.826,Y -33.337,Z -80.855,A -90.000,B 90.000,C 0.000} C_DIS
LIN {X 102.313,Y -33.335,Z -81.637,A -90.000,B 90.000,C 0.000} C_DIS
LIN {X 101.625,Y -33.339,Z -82.680,A -90.000,B 90.000,C 0.000} C_DIS
LIN {X 101.264,Y -33.341,Z -83.202,A -90.000,B 90.000,C 0.000} C_DIS
LIN {X 99.642,Y -33.348,Z -85.508,A -90.000,B 90.000,C 0.000} C_DIS
LIN {X 98.607,Y -33.352,Z -86.961,A -90.000,B 90.000,C 0.000} C_DIS
LIN {X 98.205,Y -33.355,Z -87.522,A -90.000,B 90.000,C 0.000} C_DIS
LIN {X 98.153,Y -33.362,Z -87.648,A -90.000,B 90.000,C 0.000} C_DIS
LIN {X 98.087,Y -33.385,Z -87.881,A -90.000,B 90.000,C 0.000} C_DIS
LIN {X 98.004,Y -33.420,Z -88.169,A -90.000,B 90.000,C 0.000} C_DIS
LIN {X 97.974,Y -33.443,Z -88.314,A -90.000,B 90.000,C 0.000} C_DIS
LIN {X 97.912,Y -33.498,Z -88.604,A -90.000,B 90.000,C 0.000} C_DIS
LIN {X 97.896,Y -33.509,Z -88.695,A -90.000,B 90.000,C 0.000} C_DIS
LIN {X 97.841,Y -33.527,Z -89.060,A -90.000,B 90.000,C 0.000} C_DIS
LIN {X 97.813,Y -33.539,Z -89.238,A -90.000,B 90.000,C 0.000} C_DIS
LIN {X 97.772,Y -33.545,Z -89.544,A -90.000,B 90.000,C 0.000} C_DIS
LIN {X 97.687,Y -33.572,Z -90.322,A -90.000,B 90.000,C 0.000} C_DIS
LIN {X 97.668,Y -33.577,Z -90.501,A -90.000,B 90.000,C 0.000} C_DIS
LIN {X 97.585,Y -33.588,Z -91.252,A -90.000,B 90.000,C 0.000} C_DIS
LIN {X 97.472,Y -33.605,Z -92.351,A -90.000,B 90.000,C 0.000} C_DIS
LIN {X 97.369,Y -33.622,Z -93.464,A -90.000,B 90.000,C 0.000} C_DIS
LIN {X 97.338,Y -33.626,Z -93.756,A -90.000,B 90.000,C 0.000} C_DIS
LIN {X 97.258,Y -33.629,Z -94.319,A -90.000,B 90.000,C 0.000} C_DIS
LIN {X 97.164,Y -33.638,Z -94.972,A -90.000,B 90.000,C 0.000} C_DIS
LIN {X 97.141,Y -33.641,Z -95.131,A -90.000,B 90.000,C 0.000} C_DIS
LIN {X 97.047,Y -33.631,Z -95.643,A -90.000,B 90.000,C 0.000} C_DIS
LIN {X 97.009,Y -33.626,Z -95.837,A -90.000,B 90.000,C 0.000} C_DIS
LIN {X 96.931,Y -33.628,Z -96.214,A -90.000,B 90.000,C 0.000} C_DIS
LIN {X 96.819,Y -33.637,Z -96.750,A -90.000,B 90.000,C 0.000} C_DIS
LIN {X 96.748,Y -33.628,Z -96.993,A -90.000,B 90.000,C 0.000} C_DIS
LIN {X 96.616,Y -33.616,Z -97.488,A -90.000,B 90.000,C 0.000} C_DIS
LIN {X 96.585,Y -33.616,Z -97.598,A -90.000,B 90.000,C 0.000} C_DIS
LIN {X 96.518,Y -33.621,Z -97.813,A -90.000,B 90.000,C 0.000} C_DIS
LIN {X 96.424,Y -33.621,Z -98.115,A -90.000,B 90.000,C 0.000} C_DIS
LIN {X 96.371,Y -33.620,Z -98.273,A -90.000,B 90.000,C 0.000} C_DIS
LIN {X 96.280,Y -33.610,Z -98.507,A -90.000,B 90.000,C 0.000} C_DIS
LIN {X 96.157,Y -33.601,Z -98.819,A -90.000,B 90.000,C 0.000} C_DIS
LIN {X 96.096,Y -33.599,Z -98.984,A -90.000,B 90.000,C 0.000} C_DIS
LIN {X 95.834,Y -33.618,Z -99.644,A -90.000,B 90.000,C 0.000} C_DIS
LIN {X 95.685,Y -33.631,Z -100.032,A -90.000,B 90.000,C 0.000} C_DIS
LIN {X 95.412,Y -33.677,Z -100.818,A -90.000,B 90.000,C 0.000} C_DIS
LIN {X 95.380,Y -33.680,Z -100.914,A -90.000,B 90.000,C 0.000} C_DIS
LIN {X 95.065,Y -33.737,Z -101.945,A -90.000,B 90.000,C 0.000} C_DIS
LIN {X 95.054,Y -33.739,Z -101.981,A -90.000,B 90.000,C 0.000} C_DIS
LIN {X 94.928,Y -33.739,Z -102.358,A -90.000,B 90.000,C 0.000} C_DIS
LIN {X 94.731,Y -33.762,Z -103.031,A -90.000,B 90.000,C 0.000} C_DIS
LIN {X 94.686,Y -33.769,Z -103.176,A -90.000,B 90.000,C 0.000} C_DIS
LIN {X 94.564,Y -33.778,Z -103.597,A -90.000,B 90.000,C 0.000} C_DIS
LIN {X 94.470,Y -33.805,Z -104.001,A -90.000,B 90.000,C 0.000} C_DIS
LIN {X 94.380,Y -33.809,Z -104.470,A -90.000,B 90.000,C 0.000} C_DIS
LIN {X 94.369,Y -33.822,Z -104.594,A -90.000,B 90.000,C 0.000} C_DIS
LIN {X 94.370,Y -33.820,Z -104.839,A -90.000,B 90.000,C 0.000} C_DIS
LIN {X 94.381,Y -33.798,Z -105.075,A -90.000,B 90.000,C 0.000} C_DIS
LIN {X 94.471,Y -33.789,Z -105.720,A -90.000,B 90.000,C 0.000} C_DIS
LIN {X 94.489,Y -33.785,Z -105.841,A -90.000,B 90.000,C 0.000} C_DIS
LIN {X 94.635,Y -33.780,Z -106.678,A -90.000,B 90.000,C 0.000} C_DIS
LIN {X 94.676,Y -33.785,Z -106.943,A -90.000,B 90.000,C 0.000} C_DIS
LIN {X 94.821,Y -33.786,Z -108.082,A -90.000,B 90.000,C 0.000} C_DIS
LIN {X 94.838,Y -33.790,Z -108.236,A -90.000,B 90.000,C 0.000} C_DIS
LIN {X 94.863,Y -33.790,Z -108.665,A -90.000,B 90.000,C 0.000} C_DIS
LIN {X 94.924,Y -33.802,Z -110.272,A -90.000,B 90.000,C 0.000} C_DIS
LIN {X 94.925,Y -33.802,Z -110.446,A -90.000,B 90.000,C 0.000} C_DIS
LIN {X 94.911,Y -33.812,Z -112.241,A -90.000,B 90.000,C 0.000} C_DIS
LIN {X 94.905,Y -33.811,Z -112.471,A -90.000,B 90.000,C 0.000} C_DIS
LIN {X 94.854,Y -33.830,Z -114.514,A -90.000,B 90.000,C 0.000} C_DIS
LIN {X 94.834,Y -33.836,Z -115.599,A -90.000,B 90.000,C 0.000} C_DIS
LIN {X 94.827,Y -33.839,Z -116.019,A -90.000,B 90.000,C 0.000} C_DIS
LIN {X 94.821,Y -33.841,Z -116.377,A -90.000,B 90.000,C 0.000} C_DIS
LIN {X 94.820,Y -33.845,Z -116.651,A -90.000,B 90.000,C 0.000} C_DIS
LIN {X 94.825,Y -33.846,Z -117.186,A -90.000,B 90.000,C 0.000} C_DIS
LIN {X 94.832,Y -33.858,Z -118.765,A -90.000,B 90.000,C 0.000} C_DIS
LIN {X 94.853,Y -33.861,Z -120.019,A -90.000,B 90.000,C 0.000} C_DIS
LIN {X 94.867,Y -33.865,Z -120.721,A -90.000,B 90.000,C 0.000} C_DIS
LIN {X 94.886,Y -33.865,Z -122.074,A -90.000,B 90.000,C 0.000} C_DIS
LIN {X 94.896,Y -33.867,Z -122.669,A -90.000,B 90.000,C 0.000} C_DIS
LIN {X 94.901,Y -33.866,Z -122.861,A -90.000,B 90.000,C 0.000} C_DIS
LIN {X 94.902,Y -33.864,Z -123.010,A -90.000,B 90.000,C 0.000} C_DIS
LIN {X 94.893,Y -33.866,Z -124.092,A -90.000,B 90.000,C 0.000} C_DIS
LIN {X 94.890,Y -33.869,Z -124.703,A -90.000,B 90.000,C 0.000} C_DIS
LIN {X 94.891,Y -33.867,Z -125.057,A -90.000,B 90.000,C 0.000} C_DIS
LIN {X 94.854,Y -33.867,Z -125.899,A -90.000,B 90.000,C 0.000} C_DIS
LIN {X 94.796,Y -33.873,Z -127.107,A -90.000,B 90.000,C 0.000} C_DIS
LIN {X 94.775,Y -33.870,Z -127.436,A -90.000,B 90.000,C 0.000} C_DIS
LIN {X 94.635,Y -33.880,Z -129.235,A -90.000,B 90.000,C 0.000} C_DIS
LIN {X 94.599,Y -33.880,Z -129.657,A -90.000,B 90.000,C 0.000} C_DIS
LIN {X 94.383,Y -33.892,Z -131.995,A -90.000,B 90.000,C 0.000} C_DIS
LIN {X 94.149,Y -33.900,Z -134.508,A -90.000,B 90.000,C 0.000} C_DIS
LIN {X 93.858,Y -33.902,Z -137.961,A -90.000,B 90.000,C 0.000} C_DIS
LIN {X 93.581,Y -33.901,Z -141.163,A -90.000,B 90.000,C 0.000} C_DIS
LIN {X 93.509,Y -33.903,Z -141.904,A -90.000,B 90.000,C 0.000} C_DIS
LIN {X 93.372,Y -33.902,Z -143.293,A -90.000,B 90.000,C 0.000} C_DIS
LIN {X 93.214,Y -33.900,Z -144.900,A -90.000,B 90.000,C 0.000} C_DIS
LIN {X 93.199,Y -33.901,Z -145.046,A -90.000,B 90.000,C 0.000} C_DIS
LIN {X 92.949,Y -33.900,Z -147.128,A -90.000,B 90.000,C 0.000} C_DIS
LIN {X 92.761,Y -33.897,Z -148.716,A -90.000,B 90.000,C 0.000} C_DIS
LIN {X 92.749,Y -33.898,Z -148.812,A -90.000,B 90.000,C 0.000} C_DIS
LIN {X 92.488,Y -33.893,Z -150.563,A -90.000,B 90.000,C 0.000} C_DIS
LIN {X 92.195,Y -33.892,Z -152.498,A -90.000,B 90.000,C 0.000} C_DIS
LIN {X 92.132,Y -33.886,Z -152.869,A -90.000,B 90.000,C 0.000} C_DIS
LIN {X 91.885,Y -33.882,Z -154.237,A -90.000,B 90.000,C 0.000} C_DIS
LIN {X 91.537,Y -33.881,Z -156.130,A -90.000,B 90.000,C 0.000} C_DIS
LIN {X 91.447,Y -33.876,Z -156.589,A -90.000,B 90.000,C 0.000} C_DIS
LIN {X 91.167,Y -33.872,Z -157.901,A -90.000,B 90.000,C 0.000} C_DIS
LIN {X 90.684,Y -33.872,Z -160.144,A -90.000,B 90.000,C 0.000} C_DIS
LIN {X 90.337,Y -33.869,Z -161.562,A -90.000,B 90.000,C 0.000} C_DIS
LIN {X 89.801,Y -33.870,Z -163.737,A -90.000,B 90.000,C 0.000} C_DIS
LIN {X 89.756,Y -33.869,Z -163.905,A -90.000,B 90.000,C 0.000} C_DIS
LIN {X 88.873,Y -33.870,Z -167.097,A -90.000,B 90.000,C 0.000} C_DIS
LIN {X 88.805,Y -33.871,Z -167.346,A -90.000,B 90.000,C 0.000} C_DIS
LIN {X 88.652,Y -33.866,Z -167.877,A -90.000,B 90.000,C 0.000} C_DIS
LIN {X 87.825,Y -33.869,Z -170.645,A -90.000,B 90.000,C 0.000} C_DIS
LIN {X 87.750,Y -33.870,Z -170.897,A -90.000,B 90.000,C 0.000} C_DIS
LIN {X 87.574,Y -33.867,Z -171.470,A -90.000,B 90.000,C 0.000} C_DIS
LIN {X 86.683,Y -33.870,Z -174.319,A -90.000,B 90.000,C 0.000} C_DIS
LIN {X 85.846,Y -33.867,Z -176.948,A -90.000,B 90.000,C 0.000} C_DIS
LIN {X 85.072,Y -33.868,Z -179.378,A -90.000,B 90.000,C 0.000} C_DIS
LIN {X 84.608,Y -33.861,Z -180.858,A -90.000,B 90.000,C 0.000} C_DIS
LIN {X 84.324,Y -33.860,Z -181.757,A -90.000,B 90.000,C 0.000} C_DIS
LIN {X 83.757,Y -33.847,Z -183.580,A -90.000,B 90.000,C 0.000} C_DIS
LIN {X 83.447,Y -33.847,Z -184.558,A -90.000,B 90.000,C 0.000} C_DIS
LIN {X 82.944,Y -33.834,Z -186.178,A -90.000,B 90.000,C 0.000} C_DIS
LIN {X 82.605,Y -33.833,Z -187.241,A -90.000,B 90.000,C 0.000} C_DIS
LIN {X 82.152,Y -33.822,Z -188.694,A -90.000,B 90.000,C 0.000} C_DIS
LIN {X 81.783,Y -33.823,Z -189.841,A -90.000,B 90.000,C 0.000} C_DIS
LIN {X 81.364,Y -33.815,Z -191.162,A -90.000,B 90.000,C 0.000} C_DIS
LIN {X 80.933,Y -33.817,Z -192.464,A -90.000,B 90.000,C 0.000} C_DIS
LIN {X 80.435,Y -33.812,Z -193.974,A -90.000,B 90.000,C 0.000} C_DIS
LIN {X 80.208,Y -33.814,Z -194.642,A -90.000,B 90.000,C 0.000} C_DIS
LIN {X 79.439,Y -33.813,Z -196.860,A -90.000,B 90.000,C 0.000} C_DIS
LIN {X 79.380,Y -33.812,Z -197.029,A -90.000,B 90.000,C 0.000} C_DIS
LIN {X 79.129,Y -33.816,Z -197.733,A -90.000,B 90.000,C 0.000} C_DIS
LIN {X 78.173,Y -33.816,Z -200.361,A -90.000,B 90.000,C 0.000} C_DIS
LIN {X 77.809,Y -33.821,Z -201.336,A -90.000,B 90.000,C 0.000} C_DIS
LIN {X 76.679,Y -33.823,Z -204.318,A -90.000,B 90.000,C 0.000} C_DIS
LIN {X 76.213,Y -33.830,Z -205.522,A -90.000,B 90.000,C 0.000} C_DIS
LIN {X 75.974,Y -33.830,Z -206.131,A -90.000,B 90.000,C 0.000} C_DIS
LIN {X 75.022,Y -33.833,Z -208.545,A -90.000,B 90.000,C 0.000} C_DIS
LIN {X 74.860,Y -33.834,Z -208.953,A -90.000,B 90.000,C 0.000} C_DIS
LIN {X 74.089,Y -33.844,Z -210.870,A -90.000,B 90.000,C 0.000} C_DIS
LIN {X 73.351,Y -33.846,Z -212.674,A -90.000,B 90.000,C 0.000} C_DIS
LIN {X 72.987,Y -33.848,Z -213.558,A -90.000,B 90.000,C 0.000} C_DIS
LIN {X 71.809,Y -33.864,Z -216.375,A -90.000,B 90.000,C 0.000} C_DIS
LIN {X 70.911,Y -33.868,Z -218.479,A -90.000,B 90.000,C 0.000} C_DIS
LIN {X 70.806,Y -33.867,Z -218.720,A -90.000,B 90.000,C 0.000} C_DIS
LIN {X 69.923,Y -33.873,Z -220.697,A -90.000,B 90.000,C 0.000} C_DIS
LIN {X 68.621,Y -33.892,Z -223.678,A -90.000,B 90.000,C 0.000} C_DIS
LIN {X 68.498,Y -33.891,Z -223.948,A -90.000,B 90.000,C 0.000} C_DIS
LIN {X 67.583,Y -33.901,Z -225.917,A -90.000,B 90.000,C 0.000} C_DIS
LIN {X 66.166,Y -33.926,Z -229.052,A -90.000,B 90.000,C 0.000} C_DIS
LIN {X 65.871,Y -33.924,Z -229.680,A -90.000,B 90.000,C 0.000} C_DIS
LIN {X 65.106,Y -33.940,Z -231.263,A -90.000,B 90.000,C 0.000} C_DIS
LIN {X 63.929,Y -33.969,Z -233.805,A -90.000,B 90.000,C 0.000} C_DIS
LIN {X 63.619,Y -33.976,Z -234.474,A -90.000,B 90.000,C 0.000} C_DIS
LIN {X 63.301,Y -33.974,Z -235.139,A -90.000,B 90.000,C 0.000} C_DIS
LIN {X 62.966,Y -33.984,Z -235.805,A -90.000,B 90.000,C 0.000} C_DIS
LIN {X 62.888,Y -33.985,Z -235.968,A -90.000,B 90.000,C 0.000} C_DIS
LIN {X 60.910,Y -34.047,Z -240.174,A -90.000,B 90.000,C 0.000} C_DIS
LIN {X 60.694,Y -34.060,Z -240.639,A -90.000,B 90.000,C 0.000} C_DIS
LIN {X 60.207,Y -34.084,Z -241.670,A -90.000,B 90.000,C 0.000} C_DIS
LIN {X 59.322,Y -34.123,Z -243.561,A -90.000,B 90.000,C 0.000} C_DIS
LIN {X 59.233,Y -34.131,Z -243.762,A -90.000,B 90.000,C 0.000} C_DIS
LIN {X 59.156,Y -34.132,Z -243.937,A -90.000,B 90.000,C 0.000} C_DIS
LIN {X 59.092,Y -34.133,Z -244.089,A -90.000,B 90.000,C 0.000} C_DIS
LIN {X 59.021,Y -34.130,Z -244.275,A -90.000,B 90.000,C 0.000} C_DIS
LIN {X 58.989,Y -34.127,Z -244.372,A -90.000,B 90.000,C 0.000} C_DIS
LIN {X 58.962,Y -34.120,Z -244.480,A -90.000,B 90.000,C 0.000} C_DIS
LIN {X 58.959,Y -34.117,Z -244.506,A -90.000,B 90.000,C 0.000} C_DIS
LIN {X 58.962,Y -34.109,Z -244.545,A -90.000,B 90.000,C 0.000} C_DIS
LIN {X 58.968,Y -34.105,Z -244.557,A -90.000,B 90.000,C 0.000} C_DIS
LIN {X 58.981,Y -34.098,Z -244.568,A -90.000,B 90.000,C 0.000} C_DIS
LIN {X 58.993,Y -34.093,Z -244.569,A -90.000,B 90.000,C 0.000} C_DIS
LIN {X 59.016,Y -34.085,Z -244.564,A -90.000,B 90.000,C 0.000} C_DIS
LIN {X 59.034,Y -34.080,Z -244.555,A -90.000,B 90.000,C 0.000} C_DIS
LIN {X 59.076,Y -34.067,Z -244.526,A -90.000,B 90.000,C 0.000} C_DIS
LIN {X 59.128,Y -34.054,Z -244.482,A -90.000,B 90.000,C 0.000} C_DIS
LIN {X 59.222,Y -34.033,Z -244.389,A -90.000,B 90.000,C 0.000} C_DIS
LIN {X 59.293,Y -34.017,Z -244.311,A -90.000,B 90.000,C 0.000} C_DIS
LIN {X 59.459,Y -33.984,Z -244.117,A -90.000,B 90.000,C 0.000} C_DIS
LIN {X 59.752,Y -33.930,Z -243.747,A -90.000,B 90.000,C 0.000} C_DIS
LIN {X 60.092,Y -33.871,Z -243.302,A -90.000,B 90.000,C 0.000} C_DIS
LIN {X 60.338,Y -33.830,Z -242.972,A -90.000,B 90.000,C 0.000} C_DIS
LIN {X 61.657,Y -33.614,Z -241.173,A -90.000,B 90.000,C 0.000} C_DIS
